  LIN {X 3000.007,Y -1026.300,Z -161.723,A 89.15631,B 0.00000,C 180.00000} ; release
  LIN {X 3000.007,Y -1026.300,Z 138.277,A 89.15631,B 0.00000,C 180.00000} ; retreat
  ; Step 1351, bar 2814
  LIN {X 3750.007,Y -1026.300,Z 1034.024,A 89.15631,B 0.00000,C 180.00000} ; outside
  LIN {X 3750.007,Y -1026.300,Z 88.277,A 89.15631,B 0.00000,C 180.00000} ; preinsert
  LIN {X 3750.007,Y -1026.300,Z -161.723,A 89.15631,B 0.00000,C 180.00000} ; insert
  LIN {X 3750.007,Y -1026.300,Z -161.723,A 89.15631,B 0.00000,C 180.00000} ; release
  LIN {X 3750.007,Y -1026.300,Z 138.277,A 89.15631,B 0.00000,C 180.00000} ; retreat
  ; Step 1352, bar 2817
  LIN {X 4500.007,Y -1026.300,Z 1034.024,A 89.15631,B 0.00000,C 180.00000} ; outside
  LIN {X 4500.007,Y -1026.300,Z 88.277,A 89.15631,B 0.00000,C 180.00000} ; preinsert
  LIN {X 4500.007,Y -1026.300,Z -161.723,A 89.15631,B 0.00000,C 180.00000} ; insert
  LIN {X 4500.007,Y -1026.300,Z -161.723,A 89.15631,B 0.00000,C 180.00000} ; release
  LIN {X 4500.007,Y -1026.300,Z 138.277,A 89.15631,B 0.00000,C 180.00000} ; retreat
  ; Step 1353, bar 2820
  LIN {X 5250.007,Y -1026.300,Z 1034.024,A 89.15631,B 0.00000,C 180.00000} ; outside
  LIN {X 5250.007,Y -1026.300,Z 88.277,A 89.15631,B 0.00000,C 180.00000} ; preinsert
  LIN {X 5250.007,Y -1026.300,Z -161.723,A 89.15631,B 0.00000,C 180.00000} ; insert
  LIN {X 5250.007,Y -1026.300,Z -161.723,A 89.15631,B 0.00000,C 180.00000} ; release
  LIN {X 5250.007,Y -1026.300,Z 138.277,A 89.15631,B 0.00000,C 180.00000} ; retreat
  ; Step 1354, bar 2823
  LIN {X 6000.007,Y -1026.300,Z 1034.024,A 89.15631,B 0.00000,C 180.00000} ; outside
  LIN {X 6000.007,Y -1026.300,Z 88.277,A 89.15631,B 0.00000,C 180.00000} ; preinsert
  LIN {X 6000.007,Y -1026.300,Z -161.723,A 89.15631,B 0.00000,C 180.00000} ; insert
  LIN {X 6000.007,Y -1026.300,Z -161.723,A 89.15631,B 0.00000,C 180.00000} ; release
  LIN {X 6000.007,Y -1026.300,Z 138.277,A 89.15631,B 0.00000,C 180.00000} ; retreat
  ; Step 1355, bar 2826
  LIN {X 6750.007,Y -1026.300,Z 1034.024,A 89.15631,B 0.00000,C 180.00000} ; outside
  LIN {X 6750.007,Y -1026.300,Z 88.277,A 89.15631,B 0.00000,C 180.00000} ; preinsert
  LIN {X 6750.007,Y -1026.300,Z -161.723,A 89.15631,B 0.00000,C 180.00000} ; insert
  LIN {X 6750.007,Y -1026.300,Z -161.723,A 89.15631,B 0.00000,C 180.00000} ; release
  LIN {X 6750.007,Y -1026.300,Z 138.277,A 89.15631,B 0.00000,C 180.00000} ; retreat
  ; Step 1356, bar 2829
  LIN {X 7500.007,Y -1026.300,Z 1034.024,A 89.15631,B 0.00000,C 180.00000} ; outside
  LIN {X 7500.007,Y -1026.300,Z 88.277,A 89.15631,B 0.00000,C 180.00000} ; preinsert
  LIN {X 7500.007,Y -1026.300,Z -161.723,A 89.15631,B 0.00000,C 180.00000} ; insert
  LIN {X 7500.007,Y -1026.300,Z -161.723,A 89.15631,B 0.00000,C 180.00000} ; release
  LIN {X 7500.007,Y -1026.300,Z 138.277,A 89.15631,B 0.00000,C 180.00000} ; retreat
  ; Step 1357, bar 2832
  LIN {X 8250.007,Y -1026.300,Z 1034.024,A 89.15631,B 0.00000,C 180.00000} ; outside
  LIN {X 8250.007,Y -1026.300,Z 88.277,A 89.15631,B 0.00000,C 180.00000} ; preinsert
  LIN {X 8250.007,Y -1026.300,Z -161.723,A 89.15631,B 0.00000,C 180.00000} ; insert
  LIN {X 8250.007,Y -1026.300,Z -161.723,A 89.15631,B 0.00000,C 180.00000} ; release
  LIN {X 8250.007,Y -1026.300,Z 138.277,A 89.15631,B 0.00000,C 180.00000} ; retreat
  ; Step 1358, bar 2835
  LIN {X 9000.007,Y -1026.300,Z 1034.024,A 89.15631,B 0.00000,C 180.00000} ; outside
  LIN {X 9000.007,Y -1026.300,Z 88.277,A 89.15631,B 0.00000,C 180.00000} ; preinsert
  LIN {X 9000.007,Y -1026.300,Z -161.723,A 89.15631,B 0.00000,C 180.00000} ; insert
  LIN {X 9000.007,Y -1026.300,Z -161.723,A 89.15631,B 0.00000,C 180.00000} ; release
  LIN {X 9000.007,Y -1026.300,Z 138.277,A 89.15631,B 0.00000,C 180.00000} ; retreat
  ; Step 1359, bar 2838
  LIN {X 9750.007,Y -1026.300,Z 1034.024,A 89.15631,B 0.00000,C 180.00000} ; outside
  LIN {X 9750.007,Y -1026.300,Z 88.277,A 89.15631,B 0.00000,C 180.00000} ; preinsert
  LIN {X 9750.007,Y -1026.300,Z -161.723,A 89.15631,B 0.00000,C 180.00000} ; insert
  LIN {X 9750.007,Y -1026.300,Z -161.723,A 89.15631,B 0.00000,C 180.00000} ; release
  LIN {X 9750.007,Y -1026.300,Z 138.277,A 89.15631,B 0.00000,C 180.00000} ; retreat
  ; Step 1360, bar 2841
  LIN {X 10500.007,Y -1026.300,Z 1034.024,A 89.15631,B 0.00000,C 180.00000} ; outside
  LIN {X 10500.007,Y -1026.300,Z 88.277,A 89.15631,B 0.00000,C 180.00000} ; preinsert
  LIN {X 10500.007,Y -1026.300,Z -161.723,A 89.15631,B 0.00000,C 180.00000} ; insert
  LIN {X 10500.007,Y -1026.300,Z -161.723,A 89.15631,B 0.00000,C 180.00000} ; release
  LIN {X 10500.007,Y -1026.300,Z 138.277,A 89.15631,B 0.00000,C 180.00000} ; retreat
  ; Step 1361, bar 2844
  LIN {X 11250.007,Y -1026.300,Z 1034.024,A 89.15631,B 0.00000,C 180.00000} ; outside
  LIN {X 11250.007,Y -1026.300,Z 88.277,A 89.15631,B 0.00000,C 180.00000} ; preinsert
  LIN {X 11250.007,Y -1026.300,Z -161.723,A 89.15631,B 0.00000,C 180.00000} ; insert
  LIN {X 11250.007,Y -1026.300,Z -161.723,A 89.15631,B 0.00000,C 180.00000} ; release
  LIN {X 11250.007,Y -1026.300,Z 138.277,A 89.15631,B 0.00000,C 180.00000} ; retreat
  ; Step 1362, bar 2846
  LIN {X 12000.007,Y -1026.300,Z 1034.024,A 89.15631,B 0.00000,C 180.00000} ; outside
  LIN {X 12000.007,Y -1026.300,Z 88.277,A 89.15631,B 0.00000,C 180.00000} ; preinsert
  LIN {X 12000.007,Y -1026.300,Z -161.723,A 89.15631,B 0.00000,C 180.00000} ; insert
  LIN {X 12000.007,Y -1026.300,Z -161.723,A 89.15631,B 0.00000,C 180.00000} ; release
  LIN {X 12000.007,Y -1026.300,Z 138.277,A 89.15631,B 0.00000,C 180.00000} ; retreat
  ; Step 1363, bar 2760
  LIN {X -2250.007,Y -1026.300,Z 1034.024,A 90.84369,B 0.00000,C 180.00000} ; outside
  LIN {X -2250.007,Y -1026.300,Z 88.277,A 90.84369,B 0.00000,C 180.00000} ; preinsert
  LIN {X -2250.007,Y -1026.300,Z -161.723,A 90.84369,B 0.00000,C 180.00000} ; insert
  LIN {X -2250.007,Y -1026.300,Z -161.723,A 90.84369,B 0.00000,C 180.00000} ; release
  LIN {X -2250.007,Y -1026.300,Z 138.277,A 90.84369,B 0.00000,C 180.00000} ; retreat
  ; Step 1364, bar 2763
  LIN {X -3000.007,Y -1026.300,Z 1034.024,A 90.84369,B 0.00000,C 180.00000} ; outside
  LIN {X -3000.007,Y -1026.300,Z 88.277,A 90.84369,B 0.00000,C 180.00000} ; preinsert
  LIN {X -3000.007,Y -1026.300,Z -161.723,A 90.84369,B 0.00000,C 180.00000} ; insert
  LIN {X -3000.007,Y -1026.300,Z -161.723,A 90.84369,B 0.00000,C 180.00000} ; release
  LIN {X -3000.007,Y -1026.300,Z 138.277,A 90.84369,B 0.00000,C 180.00000} ; retreat
  ; Step 1365, bar 2766
  LIN {X -3750.007,Y -1026.300,Z 1034.024,A 90.84369,B 0.00000,C 180.00000} ; outside
  LIN {X -3750.007,Y -1026.300,Z 88.277,A 90.84369,B 0.00000,C 180.00000} ; preinsert
  LIN {X -3750.007,Y -1026.300,Z -161.723,A 90.84369,B 0.00000,C 180.00000} ; insert
  LIN {X -3750.007,Y -1026.300,Z -161.723,A 90.84369,B 0.00000,C 180.00000} ; release
  LIN {X -3750.007,Y -1026.300,Z 138.277,A 90.84369,B 0.00000,C 180.00000} ; retreat
  ; Step 1366, bar 2769
  LIN {X -4500.007,Y -1026.300,Z 1034.024,A 90.84369,B 0.00000,C 180.00000} ; outside
  LIN {X -4500.007,Y -1026.300,Z 88.277,A 90.84369,B 0.00000,C 180.00000} ; preinsert
  LIN {X -4500.007,Y -1026.300,Z -161.723,A 90.84369,B 0.00000,C 180.00000} ; insert
  LIN {X -4500.007,Y -1026.300,Z -161.723,A 90.84369,B 0.00000,C 180.00000} ; release
  LIN {X -4500.007,Y -1026.300,Z 138.277,A 90.84369,B 0.00000,C 180.00000} ; retreat
  ; Step 1367, bar 2772
  LIN {X -5250.007,Y -1026.300,Z 1034.024,A 90.84369,B 0.00000,C 180.00000} ; outside
  LIN {X -5250.007,Y -1026.300,Z 88.277,A 90.84369,B 0.00000,C 180.00000} ; preinsert
  LIN {X -5250.007,Y -1026.300,Z -161.723,A 90.84369,B 0.00000,C 180.00000} ; insert
  LIN {X -5250.007,Y -1026.300,Z -161.723,A 90.84369,B 0.00000,C 180.00000} ; release
  LIN {X -5250.007,Y -1026.300,Z 138.277,A 90.84369,B 0.00000,C 180.00000} ; retreat
  ; Step 1368, bar 2775
  LIN {X -6000.007,Y -1026.300,Z 1034.024,A 90.84369,B 0.00000,C 180.00000} ; outside
  LIN {X -6000.007,Y -1026.300,Z 88.277,A 90.84369,B 0.00000,C 180.00000} ; preinsert
  LIN {X -6000.007,Y -1026.300,Z -161.723,A 90.84369,B 0.00000,C 180.00000} ; insert
  LIN {X -6000.007,Y -1026.300,Z -161.723,A 90.84369,B 0.00000,C 180.00000} ; release
  LIN {X -6000.007,Y -1026.300,Z 138.277,A 90.84369,B 0.00000,C 180.00000} ; retreat
  ; Step 1369, bar 2778
  LIN {X -6750.007,Y -1026.300,Z 1034.024,A 90.84369,B 0.00000,C 180.00000} ; outside
  LIN {X -6750.007,Y -1026.300,Z 88.277,A 90.84369,B 0.00000,C 180.00000} ; preinsert
  LIN {X -6750.007,Y -1026.300,Z -161.723,A 90.84369,B 0.00000,C 180.00000} ; insert
  LIN {X -6750.007,Y -1026.300,Z -161.723,A 90.84369,B 0.00000,C 180.00000} ; release
  LIN {X -6750.007,Y -1026.300,Z 138.277,A 90.84369,B 0.00000,C 180.00000} ; retreat
  ; Step 1370, bar 2781
  LIN {X -7500.007,Y -1026.300,Z 1034.024,A 90.84369,B 0.00000,C 180.00000} ; outside
  LIN {X -7500.007,Y -1026.300,Z 88.277,A 90.84369,B 0.00000,C 180.00000} ; preinsert
  LIN {X -7500.007,Y -1026.300,Z -161.723,A 90.84369,B 0.00000,C 180.00000} ; insert
  LIN {X -7500.007,Y -1026.300,Z -161.723,A 90.84369,B 0.00000,C 180.00000} ; release
  LIN {X -7500.007,Y -1026.300,Z 138.277,A 90.84369,B 0.00000,C 180.00000} ; retreat
  ; Step 1371, bar 2784
  LIN {X -8250.007,Y -1026.300,Z 1034.024,A 90.84369,B 0.00000,C 180.00000} ; outside
  LIN {X -8250.007,Y -1026.300,Z 88.277,A 90.84369,B 0.00000,C 180.00000} ; preinsert
  LIN {X -8250.007,Y -1026.300,Z -161.723,A 90.84369,B 0.00000,C 180.00000} ; insert
  LIN {X -8250.007,Y -1026.300,Z -161.723,A 90.84369,B 0.00000,C 180.00000} ; release
  LIN {X -8250.007,Y -1026.300,Z 138.277,A 90.84369,B 0.00000,C 180.00000} ; retreat
  ; Step 1372, bar 2787
  LIN {X -9000.007,Y -1026.300,Z 1034.024,A 90.84369,B 0.00000,C 180.00000} ; outside
  LIN {X -9000.007,Y -1026.300,Z 88.277,A 90.84369,B 0.00000,C 180.00000} ; preinsert
  LIN {X -9000.007,Y -1026.300,Z -161.723,A 90.84369,B 0.00000,C 180.00000} ; insert
  LIN {X -9000.007,Y -1026.300,Z -161.723,A 90.84369,B 0.00000,C 180.00000} ; release
  LIN {X -9000.007,Y -1026.300,Z 138.277,A 90.84369,B 0.00000,C 180.00000} ; retreat
  ; Step 1373, bar 2790
  LIN {X -9750.007,Y -1026.300,Z 1034.024,A 90.84369,B 0.00000,C 180.00000} ; outside
  LIN {X -9750.007,Y -1026.300,Z 88.277,A 90.84369,B 0.00000,C 180.00000} ; preinsert
  LIN {X -9750.007,Y -1026.300,Z -161.723,A 90.84369,B 0.00000,C 180.00000} ; insert
  LIN {X -9750.007,Y -1026.300,Z -161.723,A 90.84369,B 0.00000,C 180.00000} ; release
  LIN {X -9750.007,Y -1026.300,Z 138.277,A 90.84369,B 0.00000,C 180.00000} ; retreat
  ; Step 1374, bar 2793
  LIN {X -10500.007,Y -1026.300,Z 1034.024,A 90.84369,B 0.00000,C 180.00000} ; outside
  LIN {X -10500.007,Y -1026.300,Z 88.277,A 90.84369,B 0.00000,C 180.00000} ; preinsert
  LIN {X -10500.007,Y -1026.300,Z -161.723,A 90.84369,B 0.00000,C 180.00000} ; insert
  LIN {X -10500.007,Y -1026.300,Z -161.723,A 90.84369,B 0.00000,C 180.00000} ; release
  LIN {X -10500.007,Y -1026.300,Z 138.277,A 90.84369,B 0.00000,C 180.00000} ; retreat
  ; Step 1375, bar 2796
  LIN {X -11250.007,Y -1026.300,Z 1034.024,A 90.84369,B 0.00000,C 180.00000} ; outside
  LIN {X -11250.007,Y -1026.300,Z 88.277,A 90.84369,B 0.00000,C 180.00000} ; preinsert
  LIN {X -11250.007,Y -1026.300,Z -161.723,A 90.84369,B 0.00000,C 180.00000} ; insert
  LIN {X -11250.007,Y -1026.300,Z -161.723,A 90.84369,B 0.00000,C 180.00000} ; release
  LIN {X -11250.007,Y -1026.300,Z 138.277,A 90.84369,B 0.00000,C 180.00000} ; retreat
  ; Step 1376, bar 2798
  LIN {X -12000.007,Y -1026.300,Z 1034.024,A 90.84369,B 0.00000,C 180.00000} ; outside
  LIN {X -12000.007,Y -1026.300,Z 88.277,A 90.84369,B 0.00000,C 180.00000} ; preinsert
  LIN {X -12000.007,Y -1026.300,Z -161.723,A 90.84369,B 0.00000,C 180.00000} ; insert
  LIN {X -12000.007,Y -1026.300,Z -161.723,A 90.84369,B 0.00000,C 180.00000} ; release
  LIN {X -12000.007,Y -1026.300,Z 138.277,A 90.84369,B 0.00000,C 180.00000} ; retreat
  ; Step 1377, bar 2634
  LIN {X -12000.007,Y 1026.300,Z 1034.024,A -90.84369,B 0.00000,C -180.00000} ; outside
  LIN {X -12000.007,Y 1026.300,Z 88.277,A -90.84369,B 0.00000,C -180.00000} ; preinsert
  LIN {X -12000.007,Y 1026.300,Z -161.723,A -90.84369,B 0.00000,C -180.00000} ; insert
  LIN {X -12000.007,Y 1026.300,Z -161.723,A -90.84369,B 0.00000,C -180.00000} ; release
  LIN {X -12000.007,Y 1026.300,Z 138.277,A -90.84369,B 0.00000,C -180.00000} ; retreat
  ; Step 1378, bar 2628
  LIN {X -11250.007,Y 1026.300,Z 1034.024,A -90.84369,B 0.00000,C -180.00000} ; outside
  LIN {X -11250.007,Y 1026.300,Z 88.277,A -90.84369,B 0.00000,C -180.00000} ; preinsert
  LIN {X -11250.007,Y 1026.300,Z -161.723,A -90.84369,B 0.00000,C -180.00000} ; insert
  LIN {X -11250.007,Y 1026.300,Z -161.723,A -90.84369,B 0.00000,C -180.00000} ; release
  LIN {X -11250.007,Y 1026.300,Z 138.277,A -90.84369,B 0.00000,C -180.00000} ; retreat
  ; Step 1379, bar 2621
  LIN {X -10500.007,Y 1026.300,Z 1034.024,A -90.84369,B 0.00000,C -180.00000} ; outside
  LIN {X -10500.007,Y 1026.300,Z 88.277,A -90.84369,B 0.00000,C -180.00000} ; preinsert
  LIN {X -10500.007,Y 1026.300,Z -161.723,A -90.84369,B 0.00000,C -180.00000} ; insert
  LIN {X -10500.007,Y 1026.300,Z -161.723,A -90.84369,B 0.00000,C -180.00000} ; release
  LIN {X -10500.007,Y 1026.300,Z 138.277,A -90.84369,B 0.00000,C -180.00000} ; retreat
  ; Step 1380, bar 2614
  LIN {X -9750.007,Y 1026.300,Z 1034.024,A -90.84369,B 0.00000,C -180.00000} ; outside
  LIN {X -9750.007,Y 1026.300,Z 88.277,A -90.84369,B 0.00000,C -180.00000} ; preinsert
  LIN {X -9750.007,Y 1026.300,Z -161.723,A -90.84369,B 0.00000,C -180.00000} ; insert
  LIN {X -9750.007,Y 1026.300,Z -161.723,A -90.84369,B 0.00000,C -180.00000} ; release
  LIN {X -9750.007,Y 1026.300,Z 138.277,A -90.84369,B 0.00000,C -180.00000} ; retreat
  ; Step 1381, bar 2607
  LIN {X -9000.007,Y 1026.300,Z 1034.024,A -90.84369,B 0.00000,C -180.00000} ; outside
  LIN {X -9000.007,Y 1026.300,Z 88.277,A -90.84369,B 0.00000,C -180.00000} ; preinsert
  LIN {X -9000.007,Y 1026.300,Z -161.723,A -90.84369,B 0.00000,C -180.00000} ; insert
  LIN {X -9000.007,Y 1026.300,Z -161.723,A -90.84369,B 0.00000,C -180.00000} ; release
  LIN {X -9000.007,Y 1026.300,Z 138.277,A -90.84369,B 0.00000,C -180.00000} ; retreat
  ; Step 1382, bar 2600
  LIN {X -8250.007,Y 1026.300,Z 1034.024,A -90.84369,B 0.00000,C -180.00000} ; outside
  LIN {X -8250.007,Y 1026.300,Z 88.277,A -90.84369,B 0.00000,C -180.00000} ; preinsert
  LIN {X -8250.007,Y 1026.300,Z -161.723,A -90.84369,B 0.00000,C -180.00000} ; insert
  LIN {X -8250.007,Y 1026.300,Z -161.723,A -90.84369,B 0.00000,C -180.00000} ; release
  LIN {X -8250.007,Y 1026.300,Z 138.277,A -90.84369,B 0.00000,C -180.00000} ; retreat
  ; Step 1383, bar 2593
  LIN {X -7500.007,Y 1026.300,Z 1034.024,A -90.84369,B 0.00000,C -180.00000} ; outside
  LIN {X -7500.007,Y 1026.300,Z 88.277,A -90.84369,B 0.00000,C -180.00000} ; preinsert
  LIN {X -7500.007,Y 1026.300,Z -161.723,A -90.84369,B 0.00000,C -180.00000} ; insert
  LIN {X -7500.007,Y 1026.300,Z -161.723,A -90.84369,B 0.00000,C -180.00000} ; release
  LIN {X -7500.007,Y 1026.300,Z 138.277,A -90.84369,B 0.00000,C -180.00000} ; retreat
  ; Step 1384, bar 2586
  LIN {X -6750.007,Y 1026.300,Z 1034.024,A -90.84369,B 0.00000,C -180.00000} ; outside
  LIN {X -6750.007,Y 1026.300,Z 88.277,A -90.84369,B 0.00000,C -180.00000} ; preinsert
  LIN {X -6750.007,Y 1026.300,Z -161.723,A -90.84369,B 0.00000,C -180.00000} ; insert
  LIN {X -6750.007,Y 1026.300,Z -161.723,A -90.84369,B 0.00000,C -180.00000} ; release
  LIN {X -6750.007,Y 1026.300,Z 138.277,A -90.84369,B 0.00000,C -180.00000} ; retreat
  ; Step 1385, bar 2579
  LIN {X -6000.007,Y 1026.300,Z 1034.024,A -90.84369,B 0.00000,C -180.00000} ; outside
  LIN {X -6000.007,Y 1026.300,Z 88.277,A -90.84369,B 0.00000,C -180.00000} ; preinsert
  LIN {X -6000.007,Y 1026.300,Z -161.723,A -90.84369,B 0.00000,C -180.00000} ; insert
  LIN {X -6000.007,Y 1026.300,Z -161.723,A -90.84369,B 0.00000,C -180.00000} ; release
  LIN {X -6000.007,Y 1026.300,Z 138.277,A -90.84369,B 0.00000,C -180.00000} ; retreat
  ; Step 1386, bar 2572
  LIN {X -5250.007,Y 1026.300,Z 1034.024,A -90.84369,B 0.00000,C -180.00000} ; outside
  LIN {X -5250.007,Y 1026.300,Z 88.277,A -90.84369,B 0.00000,C -180.00000} ; preinsert
  LIN {X -5250.007,Y 1026.300,Z -161.723,A -90.84369,B 0.00000,C -180.00000} ; insert
  LIN {X -5250.007,Y 1026.300,Z -161.723,A -90.84369,B 0.00000,C -180.00000} ; release
  LIN {X -5250.007,Y 1026.300,Z 138.277,A -90.84369,B 0.00000,C -180.00000} ; retreat
  ; Step 1387, bar 2565
  LIN {X -4500.007,Y 1026.300,Z 1034.024,A -90.84369,B 0.00000,C -180.00000} ; outside
  LIN {X -4500.007,Y 1026.300,Z 88.277,A -90.84369,B 0.00000,C -180.00000} ; preinsert
  LIN {X -4500.007,Y 1026.300,Z -161.723,A -90.84369,B 0.00000,C -180.00000} ; insert
  LIN {X -4500.007,Y 1026.300,Z -161.723,A -90.84369,B 0.00000,C -180.00000} ; release
  LIN {X -4500.007,Y 1026.300,Z 138.277,A -90.84369,B 0.00000,C -180.00000} ; retreat
  ; Step 1388, bar 2558
  LIN {X -3750.007,Y 1026.300,Z 1034.024,A -90.84369,B 0.00000,C -180.00000} ; outside
  LIN {X -3750.007,Y 1026.300,Z 88.277,A -90.84369,B 0.00000,C -180.00000} ; preinsert
  LIN {X -3750.007,Y 1026.300,Z -161.723,A -90.84369,B 0.00000,C -180.00000} ; insert
  LIN {X -3750.007,Y 1026.300,Z -161.723,A -90.84369,B 0.00000,C -180.00000} ; release
  LIN {X -3750.007,Y 1026.300,Z 138.277,A -90.84369,B 0.00000,C -180.00000} ; retreat
  ; Step 1389, bar 2551
  LIN {X -3000.007,Y 1026.300,Z 1034.024,A -90.84369,B 0.00000,C -180.00000} ; outside
  LIN {X -3000.007,Y 1026.300,Z 88.277,A -90.84369,B 0.00000,C -180.00000} ; preinsert
  LIN {X -3000.007,Y 1026.300,Z -161.723,A -90.84369,B 0.00000,C -180.00000} ; insert
  LIN {X -3000.007,Y 1026.300,Z -161.723,A -90.84369,B 0.00000,C -180.00000} ; release
  LIN {X -3000.007,Y 1026.300,Z 138.277,A -90.84369,B 0.00000,C -180.00000} ; retreat
  ; Step 1390, bar 2544
  LIN {X -2250.007,Y 1026.300,Z 1034.024,A -90.84369,B 0.00000,C -180.00000} ; outside
  LIN {X -2250.007,Y 1026.300,Z 88.277,A -90.84369,B 0.00000,C -180.00000} ; preinsert
  LIN {X -2250.007,Y 1026.300,Z -161.723,A -90.84369,B 0.00000,C -180.00000} ; insert
  LIN {X -2250.007,Y 1026.300,Z -161.723,A -90.84369,B 0.00000,C -180.00000} ; release
  LIN {X -2250.007,Y 1026.300,Z 138.277,A -90.84369,B 0.00000,C -180.00000} ; retreat
  ; Step 1391, bar 2537
  LIN {X -1500.007,Y 1026.300,Z 1034.024,A -90.84369,B 0.00000,C -180.00000} ; outside
  LIN {X -1500.007,Y 1026.300,Z 88.277,A -90.84369,B 0.00000,C -180.00000} ; preinsert
  LIN {X -1500.007,Y 1026.300,Z -161.723,A -90.84369,B 0.00000,C -180.00000} ; insert
  LIN {X -1500.007,Y 1026.300,Z -161.723,A -90.84369,B 0.00000,C -180.00000} ; release
  LIN {X -1500.007,Y 1026.300,Z 138.277,A -90.84369,B 0.00000,C -180.00000} ; retreat
  ; Step 1392, bar 2530
  LIN {X -750.007,Y 1026.300,Z 1034.024,A -90.84369,B 0.00000,C -180.00000} ; outside
  LIN {X -750.007,Y 1026.300,Z 88.277,A -90.84369,B 0.00000,C -180.00000} ; preinsert
  LIN {X -750.007,Y 1026.300,Z -161.723,A -90.84369,B 0.00000,C -180.00000} ; insert
  LIN {X -750.007,Y 1026.300,Z -161.723,A -90.84369,B 0.00000,C -180.00000} ; release
  LIN {X -750.007,Y 1026.300,Z 138.277,A -90.84369,B 0.00000,C -180.00000} ; retreat
  ; Step 1393, bar 1971
  LIN {X -0.007,Y 1026.300,Z 1034.024,A -90.84369,B 0.00000,C -180.00000} ; outside
  LIN {X -0.007,Y 1026.300,Z 88.277,A -90.84369,B 0.00000,C -180.00000} ; preinsert
  LIN {X -0.007,Y 1026.300,Z -161.723,A -90.84369,B 0.00000,C -180.00000} ; insert
  LIN {X -0.007,Y 1026.300,Z -161.723,A -90.84369,B 0.00000,C -180.00000} ; release
  LIN {X -0.007,Y 1026.300,Z 138.277,A -90.84369,B 0.00000,C -180.00000} ; retreat
  ; Step 1394, bar 2640
  LIN {X 750.007,Y 1026.300,Z 1034.024,A -89.15631,B 0.00000,C 180.00000} ; outside
  LIN {X 750.007,Y 1026.300,Z 88.277,A -89.15631,B 0.00000,C 180.00000} ; preinsert
  LIN {X 750.007,Y 1026.300,Z -161.723,A -89.15631,B 0.00000,C 180.00000} ; insert
  LIN {X 750.007,Y 1026.300,Z -161.723,A -89.15631,B 0.00000,C 180.00000} ; release
  LIN {X 750.007,Y 1026.300,Z 138.277,A -89.15631,B 0.00000,C 180.00000} ; retreat
  ; Step 1395, bar 2643
  LIN {X 1500.007,Y 1026.300,Z 1034.024,A -89.15631,B 0.00000,C -180.00000} ; outside
  LIN {X 1500.007,Y 1026.300,Z 88.277,A -89.15631,B 0.00000,C -180.00000} ; preinsert
  LIN {X 1500.007,Y 1026.300,Z -161.723,A -89.15631,B 0.00000,C -180.00000} ; insert
  LIN {X 1500.007,Y 1026.300,Z -161.723,A -89.15631,B 0.00000,C -180.00000} ; release
  LIN {X 1500.007,Y 1026.300,Z 138.277,A -89.15631,B 0.00000,C -180.00000} ; retreat
  ; Step 1396, bar 2646
  LIN {X 2250.007,Y 1026.300,Z 1034.024,A -89.15631,B 0.00000,C 180.00000} ; outside
  LIN {X 2250.007,Y 1026.300,Z 88.277,A -89.15631,B 0.00000,C 180.00000} ; preinsert
  LIN {X 2250.007,Y 1026.300,Z -161.723,A -89.15631,B 0.00000,C 180.00000} ; insert
  LIN {X 2250.007,Y 1026.300,Z -161.723,A -89.15631,B 0.00000,C 180.00000} ; release
  LIN {X 2250.007,Y 1026.300,Z 138.277,A -89.15631,B 0.00000,C 180.00000} ; retreat
  ; Step 1397, bar 2649
  LIN {X 3000.007,Y 1026.300,Z 1034.024,A -89.15631,B 0.00000,C 180.00000} ; outside
  LIN {X 3000.007,Y 1026.300,Z 88.277,A -89.15631,B 0.00000,C 180.00000} ; preinsert
  LIN {X 3000.007,Y 1026.300,Z -161.723,A -89.15631,B 0.00000,C 180.00000} ; insert
  LIN {X 3000.007,Y 1026.300,Z -161.723,A -89.15631,B 0.00000,C 180.00000} ; release
  LIN {X 3000.007,Y 1026.300,Z 138.277,A -89.15631,B 0.00000,C 180.00000} ; retreat
  ; Step 1398, bar 2652
  LIN {X 3750.007,Y 1026.300,Z 1034.024,A -89.15631,B 0.00000,C 180.00000} ; outside
  LIN {X 3750.007,Y 1026.300,Z 88.277,A -89.15631,B 0.00000,C 180.00000} ; preinsert
  LIN {X 3750.007,Y 1026.300,Z -161.723,A -89.15631,B 0.00000,C 180.00000} ; insert
  LIN {X 3750.007,Y 1026.300,Z -161.723,A -89.15631,B 0.00000,C 180.00000} ; release
  LIN {X 3750.007,Y 1026.300,Z 138.277,A -89.15631,B 0.00000,C 180.00000} ; retreat
  ; Step 1399, bar 2655
  LIN {X 4500.007,Y 1026.300,Z 1034.024,A -89.15631,B 0.00000,C 180.00000} ; outside
  LIN {X 4500.007,Y 1026.300,Z 88.277,A -89.15631,B 0.00000,C 180.00000} ; preinsert
  LIN {X 4500.007,Y 1026.300,Z -161.723,A -89.15631,B 0.00000,C 180.00000} ; insert
  LIN {X 4500.007,Y 1026.300,Z -161.723,A -89.15631,B 0.00000,C 180.00000} ; release
  LIN {X 4500.007,Y 1026.300,Z 138.277,A -89.15631,B 0.00000,C 180.00000} ; retreat
  ; Step 1400, bar 2658
  LIN {X 5250.007,Y 1026.300,Z 1034.024,A -89.15631,B 0.00000,C 180.00000} ; outside
  LIN {X 5250.007,Y 1026.300,Z 88.277,A -89.15631,B 0.00000,C 180.00000} ; preinsert
  LIN {X 5250.007,Y 1026.300,Z -161.723,A -89.15631,B 0.00000,C 180.00000} ; insert
  LIN {X 5250.007,Y 1026.300,Z -161.723,A -89.15631,B 0.00000,C 180.00000} ; release
  LIN {X 5250.007,Y 1026.300,Z 138.277,A -89.15631,B 0.00000,C 180.00000} ; retreat
  ; Step 1401, bar 2661
  LIN {X 6000.007,Y 1026.300,Z 1034.024,A -89.15631,B 0.00000,C 180.00000} ; outside
  LIN {X 6000.007,Y 1026.300,Z 88.277,A -89.15631,B 0.00000,C 180.00000} ; preinsert
  LIN {X 6000.007,Y 1026.300,Z -161.723,A -89.15631,B 0.00000,C 180.00000} ; insert
  LIN {X 6000.007,Y 1026.300,Z -161.723,A -89.15631,B 0.00000,C 180.00000} ; release
  LIN {X 6000.007,Y 1026.300,Z 138.277,A -89.15631,B 0.00000,C 180.00000} ; retreat
  ; Step 1402, bar 2664
  LIN {X 6750.007,Y 1026.300,Z 1034.024,A -89.15631,B 0.00000,C 180.00000} ; outside
  LIN {X 6750.007,Y 1026.300,Z 88.277,A -89.15631,B 0.00000,C 180.00000} ; preinsert
  LIN {X 6750.007,Y 1026.300,Z -161.723,A -89.15631,B 0.00000,C 180.00000} ; insert
  LIN {X 6750.007,Y 1026.300,Z -161.723,A -89.15631,B 0.00000,C 180.00000} ; release
  LIN {X 6750.007,Y 1026.300,Z 138.277,A -89.15631,B 0.00000,C 180.00000} ; retreat
  ; Step 1403, bar 2667
  LIN {X 7500.007,Y 1026.300,Z 1034.024,A -89.15631,B 0.00000,C 180.00000} ; outside
  LIN {X 7500.007,Y 1026.300,Z 88.277,A -89.15631,B 0.00000,C 180.00000} ; preinsert
  LIN {X 7500.007,Y 1026.300,Z -161.723,A -89.15631,B 0.00000,C 180.00000} ; insert
  LIN {X 7500.007,Y 1026.300,Z -161.723,A -89.15631,B 0.00000,C 180.00000} ; release
  LIN {X 7500.007,Y 1026.300,Z 138.277,A -89.15631,B 0.00000,C 180.00000} ; retreat
  ; Step 1404, bar 2670
  LIN {X 8250.007,Y 1026.300,Z 1034.024,A -89.15631,B 0.00000,C 180.00000} ; outside
  LIN {X 8250.007,Y 1026.300,Z 88.277,A -89.15631,B 0.00000,C 180.00000} ; preinsert
  LIN {X 8250.007,Y 1026.300,Z -161.723,A -89.15631,B 0.00000,C 180.00000} ; insert
  LIN {X 8250.007,Y 1026.300,Z -161.723,A -89.15631,B 0.00000,C 180.00000} ; release
  LIN {X 8250.007,Y 1026.300,Z 138.277,A -89.15631,B 0.00000,C 180.00000} ; retreat
  ; Step 1405, bar 2673
  LIN {X 9000.007,Y 1026.300,Z 1034.024,A -89.15631,B 0.00000,C 180.00000} ; outside
  LIN {X 9000.007,Y 1026.300,Z 88.277,A -89.15631,B 0.00000,C 180.00000} ; preinsert
  LIN {X 9000.007,Y 1026.300,Z -161.723,A -89.15631,B 0.00000,C 180.00000} ; insert
  LIN {X 9000.007,Y 1026.300,Z -161.723,A -89.15631,B 0.00000,C 180.00000} ; release
  LIN {X 9000.007,Y 1026.300,Z 138.277,A -89.15631,B 0.00000,C 180.00000} ; retreat
  ; Step 1406, bar 2676
  LIN {X 9750.007,Y 1026.300,Z 1034.024,A -89.15631,B 0.00000,C 180.00000} ; outside
  LIN {X 9750.007,Y 1026.300,Z 88.277,A -89.15631,B 0.00000,C 180.00000} ; preinsert
  LIN {X 9750.007,Y 1026.300,Z -161.723,A -89.15631,B 0.00000,C 180.00000} ; insert
  LIN {X 9750.007,Y 1026.300,Z -161.723,A -89.15631,B 0.00000,C 180.00000} ; release
  LIN {X 9750.007,Y 1026.300,Z 138.277,A -89.15631,B 0.00000,C 180.00000} ; retreat
  ; Step 1407, bar 2679
  LIN {X 10500.007,Y 1026.300,Z 1034.024,A -89.15631,B 0.00000,C 180.00000} ; outside
  LIN {X 10500.007,Y 1026.300,Z 88.277,A -89.15631,B 0.00000,C 180.00000} ; preinsert
  LIN {X 10500.007,Y 1026.300,Z -161.723,A -89.15631,B 0.00000,C 180.00000} ; insert
  LIN {X 10500.007,Y 1026.300,Z -161.723,A -89.15631,B 0.00000,C 180.00000} ; release
  LIN {X 10500.007,Y 1026.300,Z 138.277,A -89.15631,B 0.00000,C 180.00000} ; retreat
  ; Step 1408, bar 2682
  LIN {X 11250.007,Y 1026.300,Z 1034.024,A -89.15631,B 0.00000,C 180.00000} ; outside
  LIN {X 11250.007,Y 1026.300,Z 88.277,A -89.15631,B 0.00000,C 180.00000} ; preinsert
  LIN {X 11250.007,Y 1026.300,Z -161.723,A -89.15631,B 0.00000,C 180.00000} ; insert
  LIN {X 11250.007,Y 1026.300,Z -161.723,A -89.15631,B 0.00000,C 180.00000} ; release
  LIN {X 11250.007,Y 1026.300,Z 138.277,A -89.15631,B 0.00000,C 180.00000} ; retreat
  ; Step 1409, bar 2684
  LIN {X 12000.007,Y 1026.300,Z 1034.024,A -89.15631,B 0.00000,C 180.00000} ; outside
  LIN {X 12000.007,Y 1026.300,Z 88.277,A -89.15631,B 0.00000,C 180.00000} ; preinsert
  LIN {X 12000.007,Y 1026.300,Z -161.723,A -89.15631,B 0.00000,C 180.00000} ; insert
  LIN {X 12000.007,Y 1026.300,Z -161.723,A -89.15631,B 0.00000,C 180.00000} ; release
  LIN {X 12000.007,Y 1026.300,Z 138.277,A -89.15631,B 0.00000,C 180.00000} ; retreat
  ; Step 1410, bar 277
  LIN {X 0.000,Y 0.000,Z 1139.371,A 0.00000,B 0.00000,C 180.00000} ; outside
  LIN {X 0.000,Y 0.000,Z 193.996,A 0.00000,B 0.00000,C 180.00000} ; preinsert
  LIN {X 0.000,Y 0.000,Z -56.004,A 0.00000,B 0.00000,C 180.00000} ; insert
  LIN {X 0.000,Y 0.000,Z -56.004,A 0.00000,B 0.00000,C 180.00000} ; release
  LIN {X 0.000,Y 0.000,Z 243.996,A 0.00000,B 0.00000,C 180.00000} ; retreat
  ; Step 1411, bar 2526
  LIN {X 16150.007,Y -2866.811,Z 1027.751,A 89.15631,B 0.00000,C 180.00000} ; outside
  LIN {X 16150.007,Y -2866.811,Z 80.465,A 89.15631,B 0.00000,C 180.00000} ; preinsert
  LIN {X 16150.007,Y -2866.811,Z -169.535,A 89.15631,B 0.00000,C 180.00000} ; insert
  LIN {X 16150.007,Y -2866.811,Z -169.535,A 89.15631,B 0.00000,C 180.00000} ; release
  LIN {X 16150.007,Y -2866.811,Z 130.465,A 89.15631,B 0.00000,C 180.00000} ; retreat
  ; Step 1412, bar 2520
  LIN {X 15550.007,Y -2866.811,Z 1027.751,A 89.15631,B 0.00000,C 180.00000} ; outside
  LIN {X 15550.007,Y -2866.811,Z 80.465,A 89.15631,B 0.00000,C 180.00000} ; preinsert
  LIN {X 15550.007,Y -2866.811,Z -169.535,A 89.15631,B 0.00000,C 180.00000} ; insert
  LIN {X 15550.007,Y -2866.811,Z -169.535,A 89.15631,B 0.00000,C 180.00000} ; release
  LIN {X 15550.007,Y -2866.811,Z 130.465,A 89.15631,B 0.00000,C 180.00000} ; retreat
  ; Step 1413, bar 2508
  LIN {X 14350.007,Y -2866.811,Z 1027.751,A 89.15631,B 0.00000,C 180.00000} ; outside
  LIN {X 14350.007,Y -2866.811,Z 80.465,A 89.15631,B 0.00000,C 180.00000} ; preinsert
  LIN {X 14350.007,Y -2866.811,Z -169.535,A 89.15631,B 0.00000,C 180.00000} ; insert
  LIN {X 14350.007,Y -2866.811,Z -169.535,A 89.15631,B 0.00000,C 180.00000} ; release
  LIN {X 14350.007,Y -2866.811,Z 130.465,A 89.15631,B 0.00000,C 180.00000} ; retreat
  ; Step 1414, bar 2514
  LIN {X 14950.007,Y -2866.811,Z 1027.751,A 89.15631,B 0.00000,C 180.00000} ; outside
  LIN {X 14950.007,Y -2866.811,Z 80.465,A 89.15631,B 0.00000,C 180.00000} ; preinsert
  LIN {X 14950.007,Y -2866.811,Z -169.535,A 89.15631,B 0.00000,C 180.00000} ; insert
  LIN {X 14950.007,Y -2866.811,Z -169.535,A 89.15631,B 0.00000,C 180.00000} ; release
  LIN {X 14950.007,Y -2866.811,Z 130.465,A 89.15631,B 0.00000,C 180.00000} ; retreat
  ; Step 1415, bar 2502
  LIN {X 13750.007,Y -2866.811,Z 1027.751,A 89.15631,B 0.00000,C 180.00000} ; outside
  LIN {X 13750.007,Y -2866.811,Z 80.465,A 89.15631,B 0.00000,C 180.00000} ; preinsert
  LIN {X 13750.007,Y -2866.811,Z -169.535,A 89.15631,B 0.00000,C 180.00000} ; insert
  LIN {X 13750.007,Y -2866.811,Z -169.535,A 89.15631,B 0.00000,C 180.00000} ; release
  LIN {X 13750.007,Y -2866.811,Z 130.465,A 89.15631,B 0.00000,C 180.00000} ; retreat
  ; Step 1416, bar 2496
  LIN {X 13150.007,Y -2866.811,Z 1027.751,A 89.15631,B 0.00000,C 180.00000} ; outside
  LIN {X 13150.007,Y -2866.811,Z 80.465,A 89.15631,B 0.00000,C 180.00000} ; preinsert
  LIN {X 13150.007,Y -2866.811,Z -169.535,A 89.15631,B 0.00000,C 180.00000} ; insert
  LIN {X 13150.007,Y -2866.811,Z -169.535,A 89.15631,B 0.00000,C 180.00000} ; release
  LIN {X 13150.007,Y -2866.811,Z 130.465,A 89.15631,B 0.00000,C 180.00000} ; retreat
  ; Step 1417, bar 2490
  LIN {X 12550.007,Y -2866.811,Z 1027.751,A 89.15631,B 0.00000,C 180.00000} ; outside
  LIN {X 12550.007,Y -2866.811,Z 80.465,A 89.15631,B 0.00000,C 180.00000} ; preinsert
  LIN {X 12550.007,Y -2866.811,Z -169.535,A 89.15631,B 0.00000,C 180.00000} ; insert
  LIN {X 12550.007,Y -2866.811,Z -169.535,A 89.15631,B 0.00000,C 180.00000} ; release
  LIN {X 12550.007,Y -2866.811,Z 130.465,A 89.15631,B 0.00000,C 180.00000} ; retreat
  ; Step 1418, bar 2485
  LIN {X 12000.007,Y -2866.811,Z 1027.751,A 89.15631,B 0.00000,C 180.00000} ; outside
  LIN {X 12000.007,Y -2866.811,Z 80.465,A 89.15631,B 0.00000,C 180.00000} ; preinsert
  LIN {X 12000.007,Y -2866.811,Z -169.535,A 89.15631,B 0.00000,C 180.00000} ; insert
  LIN {X 12000.007,Y -2866.811,Z -169.535,A 89.15631,B 0.00000,C 180.00000} ; release
  LIN {X 12000.007,Y -2866.811,Z 130.465,A 89.15631,B 0.00000,C 180.00000} ; retreat
  ; Step 1419, bar 2479
  LIN {X 11250.007,Y -2866.811,Z 1027.751,A 89.15631,B 0.00000,C 180.00000} ; outside
  LIN {X 11250.007,Y -2866.811,Z 80.465,A 89.15631,B 0.00000,C 180.00000} ; preinsert
  LIN {X 11250.007,Y -2866.811,Z -169.535,A 89.15631,B 0.00000,C 180.00000} ; insert
  LIN {X 11250.007,Y -2866.811,Z -169.535,A 89.15631,B 0.00000,C 180.00000} ; release
  LIN {X 11250.007,Y -2866.811,Z 130.465,A 89.15631,B 0.00000,C 180.00000} ; retreat
  ; Step 1420, bar 2473
  LIN {X 10500.007,Y -2866.811,Z 1027.751,A 89.15631,B 0.00000,C 180.00000} ; outside
  LIN {X 10500.007,Y -2866.811,Z 80.465,A 89.15631,B 0.00000,C 180.00000} ; preinsert
  LIN {X 10500.007,Y -2866.811,Z -169.535,A 89.15631,B 0.00000,C 180.00000} ; insert
  LIN {X 10500.007,Y -2866.811,Z -169.535,A 89.15631,B 0.00000,C 180.00000} ; release
  LIN {X 10500.007,Y -2866.811,Z 130.465,A 89.15631,B 0.00000,C 180.00000} ; retreat
  ; Step 1421, bar 2467
  LIN {X 9750.007,Y -2866.811,Z 1027.751,A 89.15631,B 0.00000,C 180.00000} ; outside
  LIN {X 9750.007,Y -2866.811,Z 80.465,A 89.15631,B 0.00000,C 180.00000} ; preinsert
  LIN {X 9750.007,Y -2866.811,Z -169.535,A 89.15631,B 0.00000,C 180.00000} ; insert
  LIN {X 9750.007,Y -2866.811,Z -169.535,A 89.15631,B 0.00000,C 180.00000} ; release
  LIN {X 9750.007,Y -2866.811,Z 130.465,A 89.15631,B 0.00000,C 180.00000} ; retreat
  ; Step 1422, bar 2461
  LIN {X 9000.007,Y -2866.811,Z 1027.751,A 89.15631,B 0.00000,C 180.00000} ; outside
  LIN {X 9000.007,Y -2866.811,Z 80.465,A 89.15631,B 0.00000,C 180.00000} ; preinsert
  LIN {X 9000.007,Y -2866.811,Z -169.535,A 89.15631,B 0.00000,C 180.00000} ; insert
  LIN {X 9000.007,Y -2866.811,Z -169.535,A 89.15631,B 0.00000,C 180.00000} ; release
  LIN {X 9000.007,Y -2866.811,Z 130.465,A 89.15631,B 0.00000,C 180.00000} ; retreat
  ; Step 1423, bar 2455
  LIN {X 8250.007,Y -2866.811,Z 1027.751,A 89.15631,B 0.00000,C 180.00000} ; outside
  LIN {X 8250.007,Y -2866.811,Z 80.465,A 89.15631,B 0.00000,C 180.00000} ; preinsert
  LIN {X 8250.007,Y -2866.811,Z -169.535,A 89.15631,B 0.00000,C 180.00000} ; insert
  LIN {X 8250.007,Y -2866.811,Z -169.535,A 89.15631,B 0.00000,C 180.00000} ; release
  LIN {X 8250.007,Y -2866.811,Z 130.465,A 89.15631,B 0.00000,C 180.00000} ; retreat
  ; Step 1424, bar 2449
  LIN {X 7500.007,Y -2866.811,Z 1027.751,A 89.15631,B 0.00000,C 180.00000} ; outside
  LIN {X 7500.007,Y -2866.811,Z 80.465,A 89.15631,B 0.00000,C 180.00000} ; preinsert
  LIN {X 7500.007,Y -2866.811,Z -169.535,A 89.15631,B 0.00000,C 180.00000} ; insert
  LIN {X 7500.007,Y -2866.811,Z -169.535,A 89.15631,B 0.00000,C 180.00000} ; release
  LIN {X 7500.007,Y -2866.811,Z 130.465,A 89.15631,B 0.00000,C 180.00000} ; retreat
  ; Step 1425, bar 2443
  LIN {X 6750.007,Y -2866.811,Z 1027.751,A 89.15631,B 0.00000,C 180.00000} ; outside
  LIN {X 6750.007,Y -2866.811,Z 80.465,A 89.15631,B 0.00000,C 180.00000} ; preinsert
  LIN {X 6750.007,Y -2866.811,Z -169.535,A 89.15631,B 0.00000,C 180.00000} ; insert
  LIN {X 6750.007,Y -2866.811,Z -169.535,A 89.15631,B 0.00000,C 180.00000} ; release
  LIN {X 6750.007,Y -2866.811,Z 130.465,A 89.15631,B 0.00000,C 180.00000} ; retreat
  ; Step 1426, bar 2437
  LIN {X 6000.007,Y -2866.811,Z 1027.751,A 89.15631,B 0.00000,C 180.00000} ; outside
  LIN {X 6000.007,Y -2866.811,Z 80.465,A 89.15631,B 0.00000,C 180.00000} ; preinsert
  LIN {X 6000.007,Y -2866.811,Z -169.535,A 89.15631,B 0.00000,C 180.00000} ; insert
  LIN {X 6000.007,Y -2866.811,Z -169.535,A 89.15631,B 0.00000,C 180.00000} ; release
  LIN {X 6000.007,Y -2866.811,Z 130.465,A 89.15631,B 0.00000,C 180.00000} ; retreat
  ; Step 1427, bar 2431
  LIN {X 5250.007,Y -2866.811,Z 1027.751,A 89.15631,B 0.00000,C 180.00000} ; outside
  LIN {X 5250.007,Y -2866.811,Z 80.465,A 89.15631,B 0.00000,C 180.00000} ; preinsert
  LIN {X 5250.007,Y -2866.811,Z -169.535,A 89.15631,B 0.00000,C 180.00000} ; insert
  LIN {X 5250.007,Y -2866.811,Z -169.535,A 89.15631,B 0.00000,C 180.00000} ; release
  LIN {X 5250.007,Y -2866.811,Z 130.465,A 89.15631,B 0.00000,C 180.00000} ; retreat
  ; Step 1428, bar 2425
  LIN {X 4500.007,Y -2866.811,Z 1027.751,A 89.15631,B 0.00000,C 180.00000} ; outside
  LIN {X 4500.007,Y -2866.811,Z 80.465,A 89.15631,B 0.00000,C 180.00000} ; preinsert
  LIN {X 4500.007,Y -2866.811,Z -169.535,A 89.15631,B 0.00000,C 180.00000} ; insert
  LIN {X 4500.007,Y -2866.811,Z -169.535,A 89.15631,B 0.00000,C 180.00000} ; release
  LIN {X 4500.007,Y -2866.811,Z 130.465,A 89.15631,B 0.00000,C 180.00000} ; retreat
  ; Step 1429, bar 2419
  LIN {X 3750.007,Y -2866.811,Z 1027.751,A 89.15631,B 0.00000,C 180.00000} ; outside
  LIN {X 3750.007,Y -2866.811,Z 80.465,A 89.15631,B 0.00000,C 180.00000} ; preinsert
  LIN {X 3750.007,Y -2866.811,Z -169.535,A 89.15631,B 0.00000,C 180.00000} ; insert
  LIN {X 3750.007,Y -2866.811,Z -169.535,A 89.15631,B 0.00000,C 180.00000} ; release
  LIN {X 3750.007,Y -2866.811,Z 130.465,A 89.15631,B 0.00000,C 180.00000} ; retreat
  ; Step 1430, bar 2413
  LIN {X 3000.007,Y -2866.811,Z 1027.751,A 89.15631,B 0.00000,C 180.00000} ; outside
  LIN {X 3000.007,Y -2866.811,Z 80.465,A 89.15631,B 0.00000,C 180.00000} ; preinsert
  LIN {X 3000.007,Y -2866.811,Z -169.535,A 89.15631,B 0.00000,C 180.00000} ; insert
  LIN {X 3000.007,Y -2866.811,Z -169.535,A 89.15631,B 0.00000,C 180.00000} ; release
  LIN {X 3000.007,Y -2866.811,Z 130.465,A 89.15631,B 0.00000,C 180.00000} ; retreat
  ; Step 1431, bar 2407
  LIN {X 2250.007,Y -2866.811,Z 1027.751,A 89.15631,B 0.00000,C 180.00000} ; outside
  LIN {X 2250.007,Y -2866.811,Z 80.465,A 89.15631,B 0.00000,C 180.00000} ; preinsert
  LIN {X 2250.007,Y -2866.811,Z -169.535,A 89.15631,B 0.00000,C 180.00000} ; insert
  LIN {X 2250.007,Y -2866.811,Z -169.535,A 89.15631,B 0.00000,C 180.00000} ; release
  LIN {X 2250.007,Y -2866.811,Z 130.465,A 89.15631,B 0.00000,C 180.00000} ; retreat
  ; Step 1432, bar 2401
  LIN {X 1500.007,Y -2866.811,Z 1027.751,A 89.15631,B 0.00000,C 180.00000} ; outside
  LIN {X 1500.007,Y -2866.811,Z 80.465,A 89.15631,B 0.00000,C 180.00000} ; preinsert
  LIN {X 1500.007,Y -2866.811,Z -169.535,A 89.15631,B 0.00000,C 180.00000} ; insert
  LIN {X 1500.007,Y -2866.811,Z -169.535,A 89.15631,B 0.00000,C 180.00000} ; release
  LIN {X 1500.007,Y -2866.811,Z 130.465,A 89.15631,B 0.00000,C 180.00000} ; retreat
  ; Step 1433, bar 2395
  LIN {X 750.007,Y -2866.811,Z 1027.751,A 89.15631,B 0.00000,C 180.00000} ; outside
  LIN {X 750.007,Y -2866.811,Z 80.465,A 89.15631,B 0.00000,C 180.00000} ; preinsert
  LIN {X 750.007,Y -2866.811,Z -169.535,A 89.15631,B 0.00000,C 180.00000} ; insert
  LIN {X 750.007,Y -2866.811,Z -169.535,A 89.15631,B 0.00000,C 180.00000} ; release
  LIN {X 750.007,Y -2866.811,Z 130.465,A 89.15631,B 0.00000,C 180.00000} ; retreat
  ; Step 1434, bar 2251
  LIN {X -0.007,Y -2866.811,Z 1027.751,A 90.84369,B 0.00000,C -180.00000} ; outside
  LIN {X -0.007,Y -2866.811,Z 80.465,A 90.84369,B 0.00000,C -180.00000} ; preinsert
  LIN {X -0.007,Y -2866.811,Z -169.535,A 90.84369,B 0.00000,C -180.00000} ; insert
  LIN {X -0.007,Y -2866.811,Z -169.535,A 90.84369,B 0.00000,C -180.00000} ; release
  LIN {X -0.007,Y -2866.811,Z 130.465,A 90.84369,B 0.00000,C -180.00000} ; retreat
  ; Step 1435, bar 2257
  LIN {X -750.007,Y -2866.811,Z 1027.751,A 90.84369,B 0.00000,C 180.00000} ; outside
  LIN {X -750.007,Y -2866.811,Z 80.465,A 90.84369,B 0.00000,C 180.00000} ; preinsert
  LIN {X -750.007,Y -2866.811,Z -169.535,A 90.84369,B 0.00000,C 180.00000} ; insert
  LIN {X -750.007,Y -2866.811,Z -169.535,A 90.84369,B 0.00000,C 180.00000} ; release
  LIN {X -750.007,Y -2866.811,Z 130.465,A 90.84369,B 0.00000,C 180.00000} ; retreat
  ; Step 1436, bar 2263
  LIN {X -1500.007,Y -2866.811,Z 1027.751,A 90.84369,B 0.00000,C 180.00000} ; outside
  LIN {X -1500.007,Y -2866.811,Z 80.465,A 90.84369,B 0.00000,C 180.00000} ; preinsert
  LIN {X -1500.007,Y -2866.811,Z -169.535,A 90.84369,B 0.00000,C 180.00000} ; insert
  LIN {X -1500.007,Y -2866.811,Z -169.535,A 90.84369,B 0.00000,C 180.00000} ; release
  LIN {X -1500.007,Y -2866.811,Z 130.465,A 90.84369,B 0.00000,C 180.00000} ; retreat
  ; Step 1437, bar 2269
  LIN {X -2250.007,Y -2866.811,Z 1027.751,A 90.84369,B 0.00000,C -180.00000} ; outside
  LIN {X -2250.007,Y -2866.811,Z 80.465,A 90.84369,B 0.00000,C -180.00000} ; preinsert
  LIN {X -2250.007,Y -2866.811,Z -169.535,A 90.84369,B 0.00000,C -180.00000} ; insert
  LIN {X -2250.007,Y -2866.811,Z -169.535,A 90.84369,B 0.00000,C -180.00000} ; release
  LIN {X -2250.007,Y -2866.811,Z 130.465,A 90.84369,B 0.00000,C -180.00000} ; retreat
  ; Step 1438, bar 2275
  LIN {X -3000.007,Y -2866.811,Z 1027.751,A 90.84369,B 0.00000,C -180.00000} ; outside
  LIN {X -3000.007,Y -2866.811,Z 80.465,A 90.84369,B 0.00000,C -180.00000} ; preinsert
  LIN {X -3000.007,Y -2866.811,Z -169.535,A 90.84369,B 0.00000,C -180.00000} ; insert
  LIN {X -3000.007,Y -2866.811,Z -169.535,A 90.84369,B 0.00000,C -180.00000} ; release
  LIN {X -3000.007,Y -2866.811,Z 130.465,A 90.84369,B 0.00000,C -180.00000} ; retreat
  ; Step 1439, bar 2281
  LIN {X -3750.007,Y -2866.811,Z 1027.751,A 90.84369,B 0.00000,C -180.00000} ; outside
  LIN {X -3750.007,Y -2866.811,Z 80.465,A 90.84369,B 0.00000,C -180.00000} ; preinsert
  LIN {X -3750.007,Y -2866.811,Z -169.535,A 90.84369,B 0.00000,C -180.00000} ; insert
  LIN {X -3750.007,Y -2866.811,Z -169.535,A 90.84369,B 0.00000,C -180.00000} ; release
  LIN {X -3750.007,Y -2866.811,Z 130.465,A 90.84369,B 0.00000,C -180.00000} ; retreat
  ; Step 1440, bar 2287
  LIN {X -4500.007,Y -2866.811,Z 1027.751,A 90.84369,B 0.00000,C -180.00000} ; outside
  LIN {X -4500.007,Y -2866.811,Z 80.465,A 90.84369,B 0.00000,C -180.00000} ; preinsert
  LIN {X -4500.007,Y -2866.811,Z -169.535,A 90.84369,B 0.00000,C -180.00000} ; insert
  LIN {X -4500.007,Y -2866.811,Z -169.535,A 90.84369,B 0.00000,C -180.00000} ; release
  LIN {X -4500.007,Y -2866.811,Z 130.465,A 90.84369,B 0.00000,C -180.00000} ; retreat
  ; Step 1441, bar 2293
  LIN {X -5250.007,Y -2866.811,Z 1027.751,A 90.84369,B 0.00000,C -180.00000} ; outside
  LIN {X -5250.007,Y -2866.811,Z 80.465,A 90.84369,B 0.00000,C -180.00000} ; preinsert
  LIN {X -5250.007,Y -2866.811,Z -169.535,A 90.84369,B 0.00000,C -180.00000} ; insert
  LIN {X -5250.007,Y -2866.811,Z -169.535,A 90.84369,B 0.00000,C -180.00000} ; release
  LIN {X -5250.007,Y -2866.811,Z 130.465,A 90.84369,B 0.00000,C -180.00000} ; retreat
  ; Step 1442, bar 2299
  LIN {X -6000.007,Y -2866.811,Z 1027.751,A 90.84369,B 0.00000,C -180.00000} ; outside
  LIN {X -6000.007,Y -2866.811,Z 80.465,A 90.84369,B 0.00000,C -180.00000} ; preinsert
  LIN {X -6000.007,Y -2866.811,Z -169.535,A 90.84369,B 0.00000,C -180.00000} ; insert
  LIN {X -6000.007,Y -2866.811,Z -169.535,A 90.84369,B 0.00000,C -180.00000} ; release
  LIN {X -6000.007,Y -2866.811,Z 130.465,A 90.84369,B 0.00000,C -180.00000} ; retreat
  ; Step 1443, bar 2305
  LIN {X -6750.007,Y -2866.811,Z 1027.751,A 90.84369,B 0.00000,C -180.00000} ; outside
  LIN {X -6750.007,Y -2866.811,Z 80.465,A 90.84369,B 0.00000,C -180.00000} ; preinsert
  LIN {X -6750.007,Y -2866.811,Z -169.535,A 90.84369,B 0.00000,C -180.00000} ; insert
  LIN {X -6750.007,Y -2866.811,Z -169.535,A 90.84369,B 0.00000,C -180.00000} ; release
  LIN {X -6750.007,Y -2866.811,Z 130.465,A 90.84369,B 0.00000,C -180.00000} ; retreat
  ; Step 1444, bar 2311
  LIN {X -7500.007,Y -2866.811,Z 1027.751,A 90.84369,B 0.00000,C -180.00000} ; outside
  LIN {X -7500.007,Y -2866.811,Z 80.465,A 90.84369,B 0.00000,C -180.00000} ; preinsert
  LIN {X -7500.007,Y -2866.811,Z -169.535,A 90.84369,B 0.00000,C -180.00000} ; insert
  LIN {X -7500.007,Y -2866.811,Z -169.535,A 90.84369,B 0.00000,C -180.00000} ; release
  LIN {X -7500.007,Y -2866.811,Z 130.465,A 90.84369,B 0.00000,C -180.00000} ; retreat
  ; Step 1445, bar 2317
  LIN {X -8250.007,Y -2866.811,Z 1027.751,A 90.84369,B 0.00000,C 180.00000} ; outside
  LIN {X -8250.007,Y -2866.811,Z 80.465,A 90.84369,B 0.00000,C 180.00000} ; preinsert
  LIN {X -8250.007,Y -2866.811,Z -169.535,A 90.84369,B 0.00000,C 180.00000} ; insert
  LIN {X -8250.007,Y -2866.811,Z -169.535,A 90.84369,B 0.00000,C 180.00000} ; release
  LIN {X -8250.007,Y -2866.811,Z 130.465,A 90.84369,B 0.00000,C 180.00000} ; retreat
  ; Step 1446, bar 2323
  LIN {X -9000.007,Y -2866.811,Z 1027.751,A 90.84369,B 0.00000,C 180.00000} ; outside
  LIN {X -9000.007,Y -2866.811,Z 80.465,A 90.84369,B 0.00000,C 180.00000} ; preinsert
  LIN {X -9000.007,Y -2866.811,Z -169.535,A 90.84369,B 0.00000,C 180.00000} ; insert
  LIN {X -9000.007,Y -2866.811,Z -169.535,A 90.84369,B 0.00000,C 180.00000} ; release
  LIN {X -9000.007,Y -2866.811,Z 130.465,A 90.84369,B 0.00000,C 180.00000} ; retreat
  ; Step 1447, bar 2329
  LIN {X -9750.007,Y -2866.811,Z 1027.751,A 90.84369,B 0.00000,C 180.00000} ; outside
  LIN {X -9750.007,Y -2866.811,Z 80.465,A 90.84369,B 0.00000,C 180.00000} ; preinsert
  LIN {X -9750.007,Y -2866.811,Z -169.535,A 90.84369,B 0.00000,C 180.00000} ; insert
  LIN {X -9750.007,Y -2866.811,Z -169.535,A 90.84369,B 0.00000,C 180.00000} ; release
  LIN {X -9750.007,Y -2866.811,Z 130.465,A 90.84369,B 0.00000,C 180.00000} ; retreat
  ; Step 1448, bar 2335
  LIN {X -10500.007,Y -2866.811,Z 1027.751,A 90.84369,B 0.00000,C 180.00000} ; outside
  LIN {X -10500.007,Y -2866.811,Z 80.465,A 90.84369,B 0.00000,C 180.00000} ; preinsert
  LIN {X -10500.007,Y -2866.811,Z -169.535,A 90.84369,B 0.00000,C 180.00000} ; insert
  LIN {X -10500.007,Y -2866.811,Z -169.535,A 90.84369,B 0.00000,C 180.00000} ; release
  LIN {X -10500.007,Y -2866.811,Z 130.465,A 90.84369,B 0.00000,C 180.00000} ; retreat
  ; Step 1449, bar 2341
  LIN {X -11250.007,Y -2866.811,Z 1027.751,A 90.84369,B 0.00000,C 180.00000} ; outside
  LIN {X -11250.007,Y -2866.811,Z 80.465,A 90.84369,B 0.00000,C 180.00000} ; preinsert
  LIN {X -11250.007,Y -2866.811,Z -169.535,A 90.84369,B 0.00000,C 180.00000} ; insert
  LIN {X -11250.007,Y -2866.811,Z -169.535,A 90.84369,B 0.00000,C 180.00000} ; release
  LIN {X -11250.007,Y -2866.811,Z 130.465,A 90.84369,B 0.00000,C 180.00000} ; retreat
  ; Step 1450, bar 2347
  LIN {X -12000.007,Y -2866.811,Z 1027.751,A 90.84369,B 0.00000,C 180.00000} ; outside
  LIN {X -12000.007,Y -2866.811,Z 80.465,A 90.84369,B 0.00000,C 180.00000} ; preinsert
  LIN {X -12000.007,Y -2866.811,Z -169.535,A 90.84369,B 0.00000,C 180.00000} ; insert
  LIN {X -12000.007,Y -2866.811,Z -169.535,A 90.84369,B 0.00000,C 180.00000} ; release
  LIN {X -12000.007,Y -2866.811,Z 130.465,A 90.84369,B 0.00000,C 180.00000} ; retreat
  ; Step 1451, bar 2352
  LIN {X -12550.007,Y -2866.811,Z 1027.751,A 90.84369,B 0.00000,C 180.00000} ; outside
  LIN {X -12550.007,Y -2866.811,Z 80.465,A 90.84369,B 0.00000,C 180.00000} ; preinsert
  LIN {X -12550.007,Y -2866.811,Z -169.535,A 90.84369,B 0.00000,C 180.00000} ; insert
  LIN {X -12550.007,Y -2866.811,Z -169.535,A 90.84369,B 0.00000,C 180.00000} ; release
  LIN {X -12550.007,Y -2866.811,Z 130.465,A 90.84369,B 0.00000,C 180.00000} ; retreat
  ; Step 1452, bar 2358
  LIN {X -13150.007,Y -2866.811,Z 1027.751,A 90.84369,B 0.00000,C 180.00000} ; outside
  LIN {X -13150.007,Y -2866.811,Z 80.465,A 90.84369,B 0.00000,C 180.00000} ; preinsert
  LIN {X -13150.007,Y -2866.811,Z -169.535,A 90.84369,B 0.00000,C 180.00000} ; insert
  LIN {X -13150.007,Y -2866.811,Z -169.535,A 90.84369,B 0.00000,C 180.00000} ; release
  LIN {X -13150.007,Y -2866.811,Z 130.465,A 90.84369,B 0.00000,C 180.00000} ; retreat
  ; Step 1453, bar 2364
  LIN {X -13750.007,Y -2866.811,Z 1027.751,A 90.84369,B 0.00000,C 180.00000} ; outside
  LIN {X -13750.007,Y -2866.811,Z 80.465,A 90.84369,B 0.00000,C 180.00000} ; preinsert
  LIN {X -13750.007,Y -2866.811,Z -169.535,A 90.84369,B 0.00000,C 180.00000} ; insert
  LIN {X -13750.007,Y -2866.811,Z -169.535,A 90.84369,B 0.00000,C 180.00000} ; release
  LIN {X -13750.007,Y -2866.811,Z 130.465,A 90.84369,B 0.00000,C 180.00000} ; retreat
  ; Step 1454, bar 2376
  LIN {X -14950.007,Y -2866.811,Z 1027.751,A 90.84369,B 0.00000,C 180.00000} ; outside
  LIN {X -14950.007,Y -2866.811,Z 80.465,A 90.84369,B 0.00000,C 180.00000} ; preinsert
  LIN {X -14950.007,Y -2866.811,Z -169.535,A 90.84369,B 0.00000,C 180.00000} ; insert
  LIN {X -14950.007,Y -2866.811,Z -169.535,A 90.84369,B 0.00000,C 180.00000} ; release
  LIN {X -14950.007,Y -2866.811,Z 130.465,A 90.84369,B 0.00000,C 180.00000} ; retreat
  ; Step 1455, bar 2370
  LIN {X -14350.007,Y -2866.811,Z 1027.751,A 90.84369,B 0.00000,C 180.00000} ; outside
  LIN {X -14350.007,Y -2866.811,Z 80.465,A 90.84369,B 0.00000,C 180.00000} ; preinsert
  LIN {X -14350.007,Y -2866.811,Z -169.535,A 90.84369,B 0.00000,C 180.00000} ; insert
  LIN {X -14350.007,Y -2866.811,Z -169.535,A 90.84369,B 0.00000,C 180.00000} ; release
  LIN {X -14350.007,Y -2866.811,Z 130.465,A 90.84369,B 0.00000,C 180.00000} ; retreat
  ; Step 1456, bar 2382
  LIN {X -15550.007,Y -2866.811,Z 1027.751,A 90.84369,B 0.00000,C 180.00000} ; outside
  LIN {X -15550.007,Y -2866.811,Z 80.465,A 90.84369,B 0.00000,C 180.00000} ; preinsert
  LIN {X -15550.007,Y -2866.811,Z -169.535,A 90.84369,B 0.00000,C 180.00000} ; insert
  LIN {X -15550.007,Y -2866.811,Z -169.535,A 90.84369,B 0.00000,C 180.00000} ; release
  LIN {X -15550.007,Y -2866.811,Z 130.465,A 90.84369,B 0.00000,C 180.00000} ; retreat
  ; Step 1457, bar 2388
  LIN {X -16150.007,Y -2866.811,Z 1027.751,A 90.84369,B 0.00000,C 180.00000} ; outside
  LIN {X -16150.007,Y -2866.811,Z 80.465,A 90.84369,B 0.00000,C 180.00000} ; preinsert
  LIN {X -16150.007,Y -2866.811,Z -169.535,A 90.84369,B 0.00000,C 180.00000} ; insert
  LIN {X -16150.007,Y -2866.811,Z -169.535,A 90.84369,B 0.00000,C 180.00000} ; release
  LIN {X -16150.007,Y -2866.811,Z 130.465,A 90.84369,B 0.00000,C 180.00000} ; retreat
  ; Step 1458, bar 2109
  LIN {X -16150.007,Y 2866.811,Z 1027.751,A -90.84369,B 0.00000,C -180.00000} ; outside
  LIN {X -16150.007,Y 2866.811,Z 80.465,A -90.84369,B 0.00000,C -180.00000} ; preinsert
  LIN {X -16150.007,Y 2866.811,Z -169.535,A -90.84369,B 0.00000,C -180.00000} ; insert
  LIN {X -16150.007,Y 2866.811,Z -169.535,A -90.84369,B 0.00000,C -180.00000} ; release
  LIN {X -16150.007,Y 2866.811,Z 130.465,A -90.84369,B 0.00000,C -180.00000} ; retreat
  ; Step 1459, bar 2103
  LIN {X -15550.007,Y 2866.811,Z 1027.751,A -90.84369,B 0.00000,C -180.00000} ; outside
  LIN {X -15550.007,Y 2866.811,Z 80.465,A -90.84369,B 0.00000,C -180.00000} ; preinsert
  LIN {X -15550.007,Y 2866.811,Z -169.535,A -90.84369,B 0.00000,C -180.00000} ; insert
  LIN {X -15550.007,Y 2866.811,Z -169.535,A -90.84369,B 0.00000,C -180.00000} ; release
  LIN {X -15550.007,Y 2866.811,Z 130.465,A -90.84369,B 0.00000,C -180.00000} ; retreat
  ; Step 1460, bar 2097
  LIN {X -14950.007,Y 2866.811,Z 1027.751,A -90.84369,B 0.00000,C -180.00000} ; outside
  LIN {X -14950.007,Y 2866.811,Z 80.465,A -90.84369,B 0.00000,C -180.00000} ; preinsert
  LIN {X -14950.007,Y 2866.811,Z -169.535,A -90.84369,B 0.00000,C -180.00000} ; insert
  LIN {X -14950.007,Y 2866.811,Z -169.535,A -90.84369,B 0.00000,C -180.00000} ; release
  LIN {X -14950.007,Y 2866.811,Z 130.465,A -90.84369,B 0.00000,C -180.00000} ; retreat
  ; Step 1461, bar 2091
  LIN {X -14350.007,Y 2866.811,Z 1027.751,A -90.84369,B 0.00000,C -180.00000} ; outside
  LIN {X -14350.007,Y 2866.811,Z 80.465,A -90.84369,B 0.00000,C -180.00000} ; preinsert
  LIN {X -14350.007,Y 2866.811,Z -169.535,A -90.84369,B 0.00000,C -180.00000} ; insert
  LIN {X -14350.007,Y 2866.811,Z -169.535,A -90.84369,B 0.00000,C -180.00000} ; release
  LIN {X -14350.007,Y 2866.811,Z 130.465,A -90.84369,B 0.00000,C -180.00000} ; retreat
  ; Step 1462, bar 2085
  LIN {X -13750.007,Y 2866.811,Z 1027.751,A -90.84369,B 0.00000,C -180.00000} ; outside
  LIN {X -13750.007,Y 2866.811,Z 80.465,A -90.84369,B 0.00000,C -180.00000} ; preinsert
  LIN {X -13750.007,Y 2866.811,Z -169.535,A -90.84369,B 0.00000,C -180.00000} ; insert
  LIN {X -13750.007,Y 2866.811,Z -169.535,A -90.84369,B 0.00000,C -180.00000} ; release
  LIN {X -13750.007,Y 2866.811,Z 130.465,A -90.84369,B 0.00000,C -180.00000} ; retreat
  ; Step 1463, bar 2079
  LIN {X -13150.007,Y 2866.811,Z 1027.751,A -90.84369,B 0.00000,C -180.00000} ; outside
  LIN {X -13150.007,Y 2866.811,Z 80.465,A -90.84369,B 0.00000,C -180.00000} ; preinsert
  LIN {X -13150.007,Y 2866.811,Z -169.535,A -90.84369,B 0.00000,C -180.00000} ; insert
  LIN {X -13150.007,Y 2866.811,Z -169.535,A -90.84369,B 0.00000,C -180.00000} ; release
  LIN {X -13150.007,Y 2866.811,Z 130.465,A -90.84369,B 0.00000,C -180.00000} ; retreat
  ; Step 1464, bar 2073
  LIN {X -12550.007,Y 2866.811,Z 1027.751,A -90.84369,B 0.00000,C -180.00000} ; outside
  LIN {X -12550.007,Y 2866.811,Z 80.465,A -90.84369,B 0.00000,C -180.00000} ; preinsert
  LIN {X -12550.007,Y 2866.811,Z -169.535,A -90.84369,B 0.00000,C -180.00000} ; insert
  LIN {X -12550.007,Y 2866.811,Z -169.535,A -90.84369,B 0.00000,C -180.00000} ; release
  LIN {X -12550.007,Y 2866.811,Z 130.465,A -90.84369,B 0.00000,C -180.00000} ; retreat
  ; Step 1465, bar 2068
  LIN {X -12000.007,Y 2866.811,Z 1027.751,A -90.84369,B 0.00000,C -180.00000} ; outside
  LIN {X -12000.007,Y 2866.811,Z 80.465,A -90.84369,B 0.00000,C -180.00000} ; preinsert
  LIN {X -12000.007,Y 2866.811,Z -169.535,A -90.84369,B 0.00000,C -180.00000} ; insert
  LIN {X -12000.007,Y 2866.811,Z -169.535,A -90.84369,B 0.00000,C -180.00000} ; release
  LIN {X -12000.007,Y 2866.811,Z 130.465,A -90.84369,B 0.00000,C -180.00000} ; retreat
  ; Step 1466, bar 2062
  LIN {X -11250.007,Y 2866.811,Z 1027.751,A -90.84369,B 0.00000,C -180.00000} ; outside
  LIN {X -11250.007,Y 2866.811,Z 80.465,A -90.84369,B 0.00000,C -180.00000} ; preinsert
  LIN {X -11250.007,Y 2866.811,Z -169.535,A -90.84369,B 0.00000,C -180.00000} ; insert
  LIN {X -11250.007,Y 2866.811,Z -169.535,A -90.84369,B 0.00000,C -180.00000} ; release
  LIN {X -11250.007,Y 2866.811,Z 130.465,A -90.84369,B 0.00000,C -180.00000} ; retreat
  ; Step 1467, bar 2056
  LIN {X -10500.007,Y 2866.811,Z 1027.751,A -90.84369,B 0.00000,C -180.00000} ; outside
  LIN {X -10500.007,Y 2866.811,Z 80.465,A -90.84369,B 0.00000,C -180.00000} ; preinsert
  LIN {X -10500.007,Y 2866.811,Z -169.535,A -90.84369,B 0.00000,C -180.00000} ; insert
  LIN {X -10500.007,Y 2866.811,Z -169.535,A -90.84369,B 0.00000,C -180.00000} ; release
  LIN {X -10500.007,Y 2866.811,Z 130.465,A -90.84369,B 0.00000,C -180.00000} ; retreat
  ; Step 1468, bar 2050
  LIN {X -9750.007,Y 2866.811,Z 1027.751,A -90.84369,B 0.00000,C -180.00000} ; outside
  LIN {X -9750.007,Y 2866.811,Z 80.465,A -90.84369,B 0.00000,C -180.00000} ; preinsert
  LIN {X -9750.007,Y 2866.811,Z -169.535,A -90.84369,B 0.00000,C -180.00000} ; insert
  LIN {X -9750.007,Y 2866.811,Z -169.535,A -90.84369,B 0.00000,C -180.00000} ; release
  LIN {X -9750.007,Y 2866.811,Z 130.465,A -90.84369,B 0.00000,C -180.00000} ; retreat
  ; Step 1469, bar 2044
  LIN {X -9000.007,Y 2866.811,Z 1027.751,A -90.84369,B 0.00000,C -180.00000} ; outside
  LIN {X -9000.007,Y 2866.811,Z 80.465,A -90.84369,B 0.00000,C -180.00000} ; preinsert
  LIN {X -9000.007,Y 2866.811,Z -169.535,A -90.84369,B 0.00000,C -180.00000} ; insert
  LIN {X -9000.007,Y 2866.811,Z -169.535,A -90.84369,B 0.00000,C -180.00000} ; release
  LIN {X -9000.007,Y 2866.811,Z 130.465,A -90.84369,B 0.00000,C -180.00000} ; retreat
  ; Step 1470, bar 2038
  LIN {X -8250.007,Y 2866.811,Z 1027.751,A -90.84369,B 0.00000,C -180.00000} ; outside
  LIN {X -8250.007,Y 2866.811,Z 80.465,A -90.84369,B 0.00000,C -180.00000} ; preinsert
  LIN {X -8250.007,Y 2866.811,Z -169.535,A -90.84369,B 0.00000,C -180.00000} ; insert
  LIN {X -8250.007,Y 2866.811,Z -169.535,A -90.84369,B 0.00000,C -180.00000} ; release
  LIN {X -8250.007,Y 2866.811,Z 130.465,A -90.84369,B 0.00000,C -180.00000} ; retreat
  ; Step 1471, bar 2032
  LIN {X -7500.007,Y 2866.811,Z 1027.751,A -90.84369,B 0.00000,C 180.00000} ; outside
  LIN {X -7500.007,Y 2866.811,Z 80.465,A -90.84369,B 0.00000,C 180.00000} ; preinsert
  LIN {X -7500.007,Y 2866.811,Z -169.535,A -90.84369,B 0.00000,C 180.00000} ; insert
  LIN {X -7500.007,Y 2866.811,Z -169.535,A -90.84369,B 0.00000,C 180.00000} ; release
  LIN {X -7500.007,Y 2866.811,Z 130.465,A -90.84369,B 0.00000,C 180.00000} ; retreat
  ; Step 1472, bar 2026
  LIN {X -6750.007,Y 2866.811,Z 1027.751,A -90.84369,B 0.00000,C 180.00000} ; outside
  LIN {X -6750.007,Y 2866.811,Z 80.465,A -90.84369,B 0.00000,C 180.00000} ; preinsert
  LIN {X -6750.007,Y 2866.811,Z -169.535,A -90.84369,B 0.00000,C 180.00000} ; insert
  LIN {X -6750.007,Y 2866.811,Z -169.535,A -90.84369,B 0.00000,C 180.00000} ; release
  LIN {X -6750.007,Y 2866.811,Z 130.465,A -90.84369,B 0.00000,C 180.00000} ; retreat
  ; Step 1473, bar 2020
  LIN {X -6000.007,Y 2866.811,Z 1027.751,A -90.84369,B 0.00000,C 180.00000} ; outside
  LIN {X -6000.007,Y 2866.811,Z 80.465,A -90.84369,B 0.00000,C 180.00000} ; preinsert
  LIN {X -6000.007,Y 2866.811,Z -169.535,A -90.84369,B 0.00000,C 180.00000} ; insert
  LIN {X -6000.007,Y 2866.811,Z -169.535,A -90.84369,B 0.00000,C 180.00000} ; release
  LIN {X -6000.007,Y 2866.811,Z 130.465,A -90.84369,B 0.00000,C 180.00000} ; retreat
  ; Step 1474, bar 2014
  LIN {X -5250.007,Y 2866.811,Z 1027.751,A -90.84369,B 0.00000,C 180.00000} ; outside
  LIN {X -5250.007,Y 2866.811,Z 80.465,A -90.84369,B 0.00000,C 180.00000} ; preinsert
  LIN {X -5250.007,Y 2866.811,Z -169.535,A -90.84369,B 0.00000,C 180.00000} ; insert
  LIN {X -5250.007,Y 2866.811,Z -169.535,A -90.84369,B 0.00000,C 180.00000} ; release
  LIN {X -5250.007,Y 2866.811,Z 130.465,A -90.84369,B 0.00000,C 180.00000} ; retreat
  ; Step 1475, bar 2008
  LIN {X -4500.007,Y 2866.811,Z 1027.751,A -90.84369,B 0.00000,C 180.00000} ; outside
  LIN {X -4500.007,Y 2866.811,Z 80.465,A -90.84369,B 0.00000,C 180.00000} ; preinsert
  LIN {X -4500.007,Y 2866.811,Z -169.535,A -90.84369,B 0.00000,C 180.00000} ; insert
  LIN {X -4500.007,Y 2866.811,Z -169.535,A -90.84369,B 0.00000,C 180.00000} ; release
  LIN {X -4500.007,Y 2866.811,Z 130.465,A -90.84369,B 0.00000,C 180.00000} ; retreat
  ; Step 1476, bar 2002
  LIN {X -3750.007,Y 2866.811,Z 1027.751,A -90.84369,B 0.00000,C 180.00000} ; outside
  LIN {X -3750.007,Y 2866.811,Z 80.465,A -90.84369,B 0.00000,C 180.00000} ; preinsert
  LIN {X -3750.007,Y 2866.811,Z -169.535,A -90.84369,B 0.00000,C 180.00000} ; insert
  LIN {X -3750.007,Y 2866.811,Z -169.535,A -90.84369,B 0.00000,C 180.00000} ; release
  LIN {X -3750.007,Y 2866.811,Z 130.465,A -90.84369,B 0.00000,C 180.00000} ; retreat
  ; Step 1477, bar 1996
  LIN {X -3000.007,Y 2866.811,Z 1027.751,A -90.84369,B 0.00000,C 180.00000} ; outside
  LIN {X -3000.007,Y 2866.811,Z 80.465,A -90.84369,B 0.00000,C 180.00000} ; preinsert
  LIN {X -3000.007,Y 2866.811,Z -169.535,A -90.84369,B 0.00000,C 180.00000} ; insert
  LIN {X -3000.007,Y 2866.811,Z -169.535,A -90.84369,B 0.00000,C 180.00000} ; release
  LIN {X -3000.007,Y 2866.811,Z 130.465,A -90.84369,B 0.00000,C 180.00000} ; retreat
  ; Step 1478, bar 1990
  LIN {X -2250.007,Y 2866.811,Z 1027.751,A -90.84369,B 0.00000,C 180.00000} ; outside
  LIN {X -2250.007,Y 2866.811,Z 80.465,A -90.84369,B 0.00000,C 180.00000} ; preinsert
  LIN {X -2250.007,Y 2866.811,Z -169.535,A -90.84369,B 0.00000,C 180.00000} ; insert
  LIN {X -2250.007,Y 2866.811,Z -169.535,A -90.84369,B 0.00000,C 180.00000} ; release
  LIN {X -2250.007,Y 2866.811,Z 130.465,A -90.84369,B 0.00000,C 180.00000} ; retreat
  ; Step 1479, bar 1984
  LIN {X -1500.007,Y 2866.811,Z 1027.751,A -90.84369,B 0.00000,C -180.00000} ; outside
  LIN {X -1500.007,Y 2866.811,Z 80.465,A -90.84369,B 0.00000,C -180.00000} ; preinsert
  LIN {X -1500.007,Y 2866.811,Z -169.535,A -90.84369,B 0.00000,C -180.00000} ; insert
  LIN {X -1500.007,Y 2866.811,Z -169.535,A -90.84369,B 0.00000,C -180.00000} ; release
  LIN {X -1500.007,Y 2866.811,Z 130.465,A -90.84369,B 0.00000,C -180.00000} ; retreat
  ; Step 1480, bar 1978
  LIN {X -750.007,Y 2866.811,Z 1027.751,A -90.84369,B 0.00000,C -180.00000} ; outside
  LIN {X -750.007,Y 2866.811,Z 80.465,A -90.84369,B 0.00000,C -180.00000} ; preinsert
  LIN {X -750.007,Y 2866.811,Z -169.535,A -90.84369,B 0.00000,C -180.00000} ; insert
  LIN {X -750.007,Y 2866.811,Z -169.535,A -90.84369,B 0.00000,C -180.00000} ; release
  LIN {X -750.007,Y 2866.811,Z 130.465,A -90.84369,B 0.00000,C -180.00000} ; retreat
  ; Step 1481, bar 1965
  LIN {X -0.007,Y 2866.811,Z 1027.751,A -90.84369,B 0.00000,C -180.00000} ; outside
  LIN {X -0.007,Y 2866.811,Z 80.465,A -90.84369,B 0.00000,C -180.00000} ; preinsert
  LIN {X -0.007,Y 2866.811,Z -169.535,A -90.84369,B 0.00000,C -180.00000} ; insert
  LIN {X -0.007,Y 2866.811,Z -169.535,A -90.84369,B 0.00000,C -180.00000} ; release
  LIN {X -0.007,Y 2866.811,Z 130.465,A -90.84369,B 0.00000,C -180.00000} ; retreat
  ; Step 1482, bar 2116
  LIN {X 750.007,Y 2866.811,Z 1027.751,A -89.15631,B 0.00000,C 180.00000} ; outside
  LIN {X 750.007,Y 2866.811,Z 80.465,A -89.15631,B 0.00000,C 180.00000} ; preinsert
  LIN {X 750.007,Y 2866.811,Z -169.535,A -89.15631,B 0.00000,C 180.00000} ; insert
  LIN {X 750.007,Y 2866.811,Z -169.535,A -89.15631,B 0.00000,C 180.00000} ; release
  LIN {X 750.007,Y 2866.811,Z 130.465,A -89.15631,B 0.00000,C 180.00000} ; retreat
  ; Step 1483, bar 2122
  LIN {X 1500.007,Y 2866.811,Z 1027.751,A -89.15631,B 0.00000,C -180.00000} ; outside
  LIN {X 1500.007,Y 2866.811,Z 80.465,A -89.15631,B 0.00000,C -180.00000} ; preinsert
  LIN {X 1500.007,Y 2866.811,Z -169.535,A -89.15631,B 0.00000,C -180.00000} ; insert
  LIN {X 1500.007,Y 2866.811,Z -169.535,A -89.15631,B 0.00000,C -180.00000} ; release
  LIN {X 1500.007,Y 2866.811,Z 130.465,A -89.15631,B 0.00000,C -180.00000} ; retreat
  ; Step 1484, bar 2128
  LIN {X 2250.007,Y 2866.811,Z 1027.751,A -89.15631,B 0.00000,C 180.00000} ; outside
  LIN {X 2250.007,Y 2866.811,Z 80.465,A -89.15631,B 0.00000,C 180.00000} ; preinsert
  LIN {X 2250.007,Y 2866.811,Z -169.535,A -89.15631,B 0.00000,C 180.00000} ; insert
  LIN {X 2250.007,Y 2866.811,Z -169.535,A -89.15631,B 0.00000,C 180.00000} ; release
  LIN {X 2250.007,Y 2866.811,Z 130.465,A -89.15631,B 0.00000,C 180.00000} ; retreat
  ; Step 1485, bar 2134
  LIN {X 3000.007,Y 2866.811,Z 1027.751,A -89.15631,B 0.00000,C 180.00000} ; outside
  LIN {X 3000.007,Y 2866.811,Z 80.465,A -89.15631,B 0.00000,C 180.00000} ; preinsert
  LIN {X 3000.007,Y 2866.811,Z -169.535,A -89.15631,B 0.00000,C 180.00000} ; insert
  LIN {X 3000.007,Y 2866.811,Z -169.535,A -89.15631,B 0.00000,C 180.00000} ; release
  LIN {X 3000.007,Y 2866.811,Z 130.465,A -89.15631,B 0.00000,C 180.00000} ; retreat
  ; Step 1486, bar 2140
  LIN {X 3750.007,Y 2866.811,Z 1027.751,A -89.15631,B 0.00000,C 180.00000} ; outside
  LIN {X 3750.007,Y 2866.811,Z 80.465,A -89.15631,B 0.00000,C 180.00000} ; preinsert
  LIN {X 3750.007,Y 2866.811,Z -169.535,A -89.15631,B 0.00000,C 180.00000} ; insert
  LIN {X 3750.007,Y 2866.811,Z -169.535,A -89.15631,B 0.00000,C 180.00000} ; release
  LIN {X 3750.007,Y 2866.811,Z 130.465,A -89.15631,B 0.00000,C 180.00000} ; retreat
  ; Step 1487, bar 2146
  LIN {X 4500.007,Y 2866.811,Z 1027.751,A -89.15631,B 0.00000,C 180.00000} ; outside
  LIN {X 4500.007,Y 2866.811,Z 80.465,A -89.15631,B 0.00000,C 180.00000} ; preinsert
  LIN {X 4500.007,Y 2866.811,Z -169.535,A -89.15631,B 0.00000,C 180.00000} ; insert
  LIN {X 4500.007,Y 2866.811,Z -169.535,A -89.15631,B 0.00000,C 180.00000} ; release
  LIN {X 4500.007,Y 2866.811,Z 130.465,A -89.15631,B 0.00000,C 180.00000} ; retreat
  ; Step 1488, bar 2152
  LIN {X 5250.007,Y 2866.811,Z 1027.751,A -89.15631,B 0.00000,C 180.00000} ; outside
  LIN {X 5250.007,Y 2866.811,Z 80.465,A -89.15631,B 0.00000,C 180.00000} ; preinsert
  LIN {X 5250.007,Y 2866.811,Z -169.535,A -89.15631,B 0.00000,C 180.00000} ; insert
  LIN {X 5250.007,Y 2866.811,Z -169.535,A -89.15631,B 0.00000,C 180.00000} ; release
  LIN {X 5250.007,Y 2866.811,Z 130.465,A -89.15631,B 0.00000,C 180.00000} ; retreat
  ; Step 1489, bar 2158
  LIN {X 6000.007,Y 2866.811,Z 1027.751,A -89.15631,B 0.00000,C 180.00000} ; outside
  LIN {X 6000.007,Y 2866.811,Z 80.465,A -89.15631,B 0.00000,C 180.00000} ; preinsert
  LIN {X 6000.007,Y 2866.811,Z -169.535,A -89.15631,B 0.00000,C 180.00000} ; insert
  LIN {X 6000.007,Y 2866.811,Z -169.535,A -89.15631,B 0.00000,C 180.00000} ; release
  LIN {X 6000.007,Y 2866.811,Z 130.465,A -89.15631,B 0.00000,C 180.00000} ; retreat
  ; Step 1490, bar 2164
  LIN {X 6750.007,Y 2866.811,Z 1027.751,A -89.15631,B 0.00000,C 180.00000} ; outside
  LIN {X 6750.007,Y 2866.811,Z 80.465,A -89.15631,B 0.00000,C 180.00000} ; preinsert
  LIN {X 6750.007,Y 2866.811,Z -169.535,A -89.15631,B 0.00000,C 180.00000} ; insert
  LIN {X 6750.007,Y 2866.811,Z -169.535,A -89.15631,B 0.00000,C 180.00000} ; release
  LIN {X 6750.007,Y 2866.811,Z 130.465,A -89.15631,B 0.00000,C 180.00000} ; retreat
  ; Step 1491, bar 2170
  LIN {X 7500.007,Y 2866.811,Z 1027.751,A -89.15631,B 0.00000,C 180.00000} ; outside
  LIN {X 7500.007,Y 2866.811,Z 80.465,A -89.15631,B 0.00000,C 180.00000} ; preinsert
  LIN {X 7500.007,Y 2866.811,Z -169.535,A -89.15631,B 0.00000,C 180.00000} ; insert
  LIN {X 7500.007,Y 2866.811,Z -169.535,A -89.15631,B 0.00000,C 180.00000} ; release
  LIN {X 7500.007,Y 2866.811,Z 130.465,A -89.15631,B 0.00000,C 180.00000} ; retreat
  ; Step 1492, bar 2176
  LIN {X 8250.007,Y 2866.811,Z 1027.751,A -89.15631,B 0.00000,C 180.00000} ; outside
  LIN {X 8250.007,Y 2866.811,Z 80.465,A -89.15631,B 0.00000,C 180.00000} ; preinsert
  LIN {X 8250.007,Y 2866.811,Z -169.535,A -89.15631,B 0.00000,C 180.00000} ; insert
  LIN {X 8250.007,Y 2866.811,Z -169.535,A -89.15631,B 0.00000,C 180.00000} ; release
  LIN {X 8250.007,Y 2866.811,Z 130.465,A -89.15631,B 0.00000,C 180.00000} ; retreat
  ; Step 1493, bar 2182
  LIN {X 9000.007,Y 2866.811,Z 1027.751,A -89.15631,B 0.00000,C 180.00000} ; outside
  LIN {X 9000.007,Y 2866.811,Z 80.465,A -89.15631,B 0.00000,C 180.00000} ; preinsert
  LIN {X 9000.007,Y 2866.811,Z -169.535,A -89.15631,B 0.00000,C 180.00000} ; insert
  LIN {X 9000.007,Y 2866.811,Z -169.535,A -89.15631,B 0.00000,C 180.00000} ; release
  LIN {X 9000.007,Y 2866.811,Z 130.465,A -89.15631,B 0.00000,C 180.00000} ; retreat
  ; Step 1494, bar 2188
  LIN {X 9750.007,Y 2866.811,Z 1027.751,A -89.15631,B 0.00000,C 180.00000} ; outside
  LIN {X 9750.007,Y 2866.811,Z 80.465,A -89.15631,B 0.00000,C 180.00000} ; preinsert
  LIN {X 9750.007,Y 2866.811,Z -169.535,A -89.15631,B 0.00000,C 180.00000} ; insert
  LIN {X 9750.007,Y 2866.811,Z -169.535,A -89.15631,B 0.00000,C 180.00000} ; release
  LIN {X 9750.007,Y 2866.811,Z 130.465,A -89.15631,B 0.00000,C 180.00000} ; retreat
  ; Step 1495, bar 2194
  LIN {X 10500.007,Y 2866.811,Z 1027.751,A -89.15631,B 0.00000,C 180.00000} ; outside
  LIN {X 10500.007,Y 2866.811,Z 80.465,A -89.15631,B 0.00000,C 180.00000} ; preinsert
  LIN {X 10500.007,Y 2866.811,Z -169.535,A -89.15631,B 0.00000,C 180.00000} ; insert
  LIN {X 10500.007,Y 2866.811,Z -169.535,A -89.15631,B 0.00000,C 180.00000} ; release
  LIN {X 10500.007,Y 2866.811,Z 130.465,A -89.15631,B 0.00000,C 180.00000} ; retreat
  ; Step 1496, bar 2200
  LIN {X 11250.007,Y 2866.811,Z 1027.751,A -89.15631,B 0.00000,C 180.00000} ; outside
  LIN {X 11250.007,Y 2866.811,Z 80.465,A -89.15631,B 0.00000,C 180.00000} ; preinsert
  LIN {X 11250.007,Y 2866.811,Z -169.535,A -89.15631,B 0.00000,C 180.00000} ; insert
  LIN {X 11250.007,Y 2866.811,Z -169.535,A -89.15631,B 0.00000,C 180.00000} ; release
  LIN {X 11250.007,Y 2866.811,Z 130.465,A -89.15631,B 0.00000,C 180.00000} ; retreat
  ; Step 1497, bar 2206
  LIN {X 12000.007,Y 2866.811,Z 1027.751,A -89.15631,B 0.00000,C 180.00000} ; outside
  LIN {X 12000.007,Y 2866.811,Z 80.465,A -89.15631,B 0.00000,C 180.00000} ; preinsert
  LIN {X 12000.007,Y 2866.811,Z -169.535,A -89.15631,B 0.00000,C 180.00000} ; insert
  LIN {X 12000.007,Y 2866.811,Z -169.535,A -89.15631,B 0.00000,C 180.00000} ; release
  LIN {X 12000.007,Y 2866.811,Z 130.465,A -89.15631,B 0.00000,C 180.00000} ; retreat
  ; Step 1498, bar 2211
  LIN {X 12550.007,Y 2866.811,Z 1027.751,A -89.15631,B 0.00000,C 180.00000} ; outside
  LIN {X 12550.007,Y 2866.811,Z 80.465,A -89.15631,B 0.00000,C 180.00000} ; preinsert
  LIN {X 12550.007,Y 2866.811,Z -169.535,A -89.15631,B 0.00000,C 180.00000} ; insert
  LIN {X 12550.007,Y 2866.811,Z -169.535,A -89.15631,B 0.00000,C 180.00000} ; release
  LIN {X 12550.007,Y 2866.811,Z 130.465,A -89.15631,B 0.00000,C 180.00000} ; retreat
  ; Step 1499, bar 2217
  LIN {X 13150.007,Y 2866.811,Z 1027.751,A -89.15631,B 0.00000,C 180.00000} ; outside
  LIN {X 13150.007,Y 2866.811,Z 80.465,A -89.15631,B 0.00000,C 180.00000} ; preinsert
  LIN {X 13150.007,Y 2866.811,Z -169.535,A -89.15631,B 0.00000,C 180.00000} ; insert
  LIN {X 13150.007,Y 2866.811,Z -169.535,A -89.15631,B 0.00000,C 180.00000} ; release
  LIN {X 13150.007,Y 2866.811,Z 130.465,A -89.15631,B 0.00000,C 180.00000} ; retreat
  ; Step 1500, bar 2223
  LIN {X 13750.007,Y 2866.811,Z 1027.751,A -89.15631,B 0.00000,C 180.00000} ; outside
  LIN {X 13750.007,Y 2866.811,Z 80.465,A -89.15631,B 0.00000,C 180.00000} ; preinsert
  LIN {X 13750.007,Y 2866.811,Z -169.535,A -89.15631,B 0.00000,C 180.00000} ; insert
  LIN {X 13750.007,Y 2866.811,Z -169.535,A -89.15631,B 0.00000,C 180.00000} ; release
  LIN {X 13750.007,Y 2866.811,Z 130.465,A -89.15631,B 0.00000,C 180.00000} ; retreat
  ; Step 1501, bar 2229
  LIN {X 14350.007,Y 2866.811,Z 1027.751,A -89.15631,B 0.00000,C 180.00000} ; outside
  LIN {X 14350.007,Y 2866.811,Z 80.465,A -89.15631,B 0.00000,C 180.00000} ; preinsert
  LIN {X 14350.007,Y 2866.811,Z -169.535,A -89.15631,B 0.00000,C 180.00000} ; insert
  LIN {X 14350.007,Y 2866.811,Z -169.535,A -89.15631,B 0.00000,C 180.00000} ; release
  LIN {X 14350.007,Y 2866.811,Z 130.465,A -89.15631,B 0.00000,C 180.00000} ; retreat
  ; Step 1502, bar 2235
  LIN {X 14950.007,Y 2866.811,Z 1027.751,A -89.15631,B 0.00000,C 180.00000} ; outside
  LIN {X 14950.007,Y 2866.811,Z 80.465,A -89.15631,B 0.00000,C 180.00000} ; preinsert
  LIN {X 14950.007,Y 2866.811,Z -169.535,A -89.15631,B 0.00000,C 180.00000} ; insert
  LIN {X 14950.007,Y 2866.811,Z -169.535,A -89.15631,B 0.00000,C 180.00000} ; release
  LIN {X 14950.007,Y 2866.811,Z 130.465,A -89.15631,B 0.00000,C 180.00000} ; retreat
  ; Step 1503, bar 2241
  LIN {X 15550.007,Y 2866.811,Z 1027.751,A -89.15631,B 0.00000,C 180.00000} ; outside
  LIN {X 15550.007,Y 2866.811,Z 80.465,A -89.15631,B 0.00000,C 180.00000} ; preinsert
  LIN {X 15550.007,Y 2866.811,Z -169.535,A -89.15631,B 0.00000,C 180.00000} ; insert
  LIN {X 15550.007,Y 2866.811,Z -169.535,A -89.15631,B 0.00000,C 180.00000} ; release
  LIN {X 15550.007,Y 2866.811,Z 130.465,A -89.15631,B 0.00000,C 180.00000} ; retreat
  ; Step 1504, bar 2247
  LIN {X 16150.007,Y 2866.811,Z 1027.751,A -89.15631,B 0.00000,C 180.00000} ; outside
  LIN {X 16150.007,Y 2866.811,Z 80.465,A -89.15631,B 0.00000,C 180.00000} ; preinsert
  LIN {X 16150.007,Y 2866.811,Z -169.535,A -89.15631,B 0.00000,C 180.00000} ; insert
  LIN {X 16150.007,Y 2866.811,Z -169.535,A -89.15631,B 0.00000,C 180.00000} ; release
  LIN {X 16150.007,Y 2866.811,Z 130.465,A -89.15631,B 0.00000,C 180.00000} ; retreat
  ; Step 1505, bar 3050
  LIN {X -16049.996,Y -1026.029,Z 973.273,A -172.46345,B 0.00000,C -180.00000} ; outside
  LIN {X -16049.996,Y -1026.029,Z 17.643,A -172.46345,B 0.00000,C -180.00000} ; preinsert
  LIN {X -16049.996,Y -1026.029,Z -232.357,A -172.46345,B 0.00000,C -180.00000} ; insert
  LIN {X -16049.996,Y -1026.029,Z -232.357,A -172.46345,B 0.00000,C -180.00000} ; release
  LIN {X -16049.996,Y -1026.029,Z 67.643,A -172.46345,B 0.00000,C -180.00000} ; retreat
  ; Step 1506, bar 3045
  LIN {X -15649.996,Y -1026.029,Z 973.273,A -172.46345,B 0.00000,C -180.00000} ; outside
  LIN {X -15649.996,Y -1026.029,Z 17.643,A -172.46345,B 0.00000,C -180.00000} ; preinsert
  LIN {X -15649.996,Y -1026.029,Z -232.357,A -172.46345,B 0.00000,C -180.00000} ; insert
  LIN {X -15649.996,Y -1026.029,Z -232.357,A -172.46345,B 0.00000,C -180.00000} ; release
  LIN {X -15649.996,Y -1026.029,Z 67.643,A -172.46345,B 0.00000,C -180.00000} ; retreat
  ; Step 1507, bar 3040
  LIN {X -15249.996,Y -1026.029,Z 973.273,A -172.46345,B 0.00000,C -180.00000} ; outside
  LIN {X -15249.996,Y -1026.029,Z 17.643,A -172.46345,B 0.00000,C -180.00000} ; preinsert
  LIN {X -15249.996,Y -1026.029,Z -232.357,A -172.46345,B 0.00000,C -180.00000} ; insert
  LIN {X -15249.996,Y -1026.029,Z -232.357,A -172.46345,B 0.00000,C -180.00000} ; release
  LIN {X -15249.996,Y -1026.029,Z 67.643,A -172.46345,B 0.00000,C -180.00000} ; retreat
  ; Step 1508, bar 3055
  LIN {X 15249.996,Y 1026.029,Z 973.273,A 7.53655,B 0.00000,C 180.00000} ; outside
  LIN {X 15249.996,Y 1026.029,Z 17.643,A 7.53655,B 0.00000,C 180.00000} ; preinsert
  LIN {X 15249.996,Y 1026.029,Z -232.357,A 7.53655,B 0.00000,C 180.00000} ; insert
  LIN {X 15249.996,Y 1026.029,Z -232.357,A 7.53655,B 0.00000,C 180.00000} ; release
  LIN {X 15249.996,Y 1026.029,Z 67.643,A 7.53655,B 0.00000,C 180.00000} ; retreat
  ; Step 1509, bar 3061
  LIN {X 15649.996,Y 1026.029,Z 973.273,A 7.53655,B 0.00000,C 180.00000} ; outside
  LIN {X 15649.996,Y 1026.029,Z 17.643,A 7.53655,B 0.00000,C 180.00000} ; preinsert
  LIN {X 15649.996,Y 1026.029,Z -232.357,A 7.53655,B 0.00000,C 180.00000} ; insert
  LIN {X 15649.996,Y 1026.029,Z -232.357,A 7.53655,B 0.00000,C 180.00000} ; release
  LIN {X 15649.996,Y 1026.029,Z 67.643,A 7.53655,B 0.00000,C 180.00000} ; retreat
  ; Step 1510, bar 3067
  LIN {X 16049.996,Y 1026.029,Z 973.273,A 7.53655,B 0.00000,C 180.00000} ; outside
  LIN {X 16049.996,Y 1026.029,Z 17.643,A 7.53655,B 0.00000,C 180.00000} ; preinsert
  LIN {X 16049.996,Y 1026.029,Z -232.357,A 7.53655,B 0.00000,C 180.00000} ; insert
  LIN {X 16049.996,Y 1026.029,Z -232.357,A 7.53655,B 0.00000,C 180.00000} ; release
  LIN {X 16049.996,Y 1026.029,Z 67.643,A 7.53655,B 0.00000,C 180.00000} ; retreat
  ; Step 1511, bar 3073
  LIN {X 15249.996,Y -1026.029,Z 973.274,A -7.53655,B 0.00000,C 180.00000} ; outside
  LIN {X 15249.996,Y -1026.029,Z 17.643,A -7.53655,B 0.00000,C 180.00000} ; preinsert
  LIN {X 15249.996,Y -1026.029,Z -232.357,A -7.53655,B 0.00000,C 180.00000} ; insert
  LIN {X 15249.996,Y -1026.029,Z -232.357,A -7.53655,B 0.00000,C 180.00000} ; release
  LIN {X 15249.996,Y -1026.029,Z 67.643,A -7.53655,B 0.00000,C 180.00000} ; retreat
  ; Step 1512, bar 3078
  LIN {X 15649.996,Y -1026.029,Z 973.274,A -7.53655,B 0.00000,C 180.00000} ; outside
  LIN {X 15649.996,Y -1026.029,Z 17.643,A -7.53655,B 0.00000,C 180.00000} ; preinsert
  LIN {X 15649.996,Y -1026.029,Z -232.357,A -7.53655,B 0.00000,C 180.00000} ; insert
  LIN {X 15649.996,Y -1026.029,Z -232.357,A -7.53655,B 0.00000,C 180.00000} ; release
  LIN {X 15649.996,Y -1026.029,Z 67.643,A -7.53655,B 0.00000,C 180.00000} ; retreat
  ; Step 1513, bar 3083
  LIN {X 16049.996,Y -1026.029,Z 973.274,A -7.53655,B 0.00000,C 180.00000} ; outside
  LIN {X 16049.996,Y -1026.029,Z 17.643,A -7.53655,B 0.00000,C 180.00000} ; preinsert
  LIN {X 16049.996,Y -1026.029,Z -232.357,A -7.53655,B 0.00000,C 180.00000} ; insert
  LIN {X 16049.996,Y -1026.029,Z -232.357,A -7.53655,B 0.00000,C 180.00000} ; release
  LIN {X 16049.996,Y -1026.029,Z 67.643,A -7.53655,B 0.00000,C 180.00000} ; retreat
  ; Step 1514, bar 3034
  LIN {X -16049.996,Y 1026.029,Z 973.274,A 172.46345,B 0.00000,C 180.00000} ; outside
  LIN {X -16049.996,Y 1026.029,Z 17.643,A 172.46345,B 0.00000,C 180.00000} ; preinsert
  LIN {X -16049.996,Y 1026.029,Z -232.357,A 172.46345,B 0.00000,C 180.00000} ; insert
  LIN {X -16049.996,Y 1026.029,Z -232.357,A 172.46345,B 0.00000,C 180.00000} ; release
  LIN {X -16049.996,Y 1026.029,Z 67.643,A 172.46345,B 0.00000,C 180.00000} ; retreat
  ; Step 1515, bar 3028
  LIN {X -15649.996,Y 1026.029,Z 973.274,A 172.46345,B 0.00000,C 180.00000} ; outside
  LIN {X -15649.996,Y 1026.029,Z 17.643,A 172.46345,B 0.00000,C 180.00000} ; preinsert
  LIN {X -15649.996,Y 1026.029,Z -232.357,A 172.46345,B 0.00000,C 180.00000} ; insert
  LIN {X -15649.996,Y 1026.029,Z -232.357,A 172.46345,B 0.00000,C 180.00000} ; release
  LIN {X -15649.996,Y 1026.029,Z 67.643,A 172.46345,B 0.00000,C 180.00000} ; retreat
  ; Step 1516, bar 3022
  LIN {X -15249.996,Y 1026.029,Z 973.274,A 172.46345,B 0.00000,C 180.00000} ; outside
  LIN {X -15249.996,Y 1026.029,Z 17.643,A 172.46345,B 0.00000,C 180.00000} ; preinsert
  LIN {X -15249.996,Y 1026.029,Z -232.357,A 172.46345,B 0.00000,C 180.00000} ; insert
  LIN {X -15249.996,Y 1026.029,Z -232.357,A 172.46345,B 0.00000,C 180.00000} ; release
  LIN {X -15249.996,Y 1026.029,Z 67.643,A 172.46345,B 0.00000,C 180.00000} ; retreat
  ; Step 1517, bar 2522
  LIN {X 15849.916,Y -3131.796,Z 1047.576,A 92.55766,B 0.00000,C -180.00000} ; outside
  LIN {X 15849.916,Y -3131.796,Z 96.905,A 92.55766,B 0.00000,C -180.00000} ; preinsert
  LIN {X 15849.916,Y -3131.796,Z -153.095,A 92.55766,B 0.00000,C -180.00000} ; insert
  LIN {X 15849.916,Y -3131.796,Z -153.095,A 92.55766,B 0.00000,C -180.00000} ; release
  LIN {X 15849.916,Y -3131.796,Z 146.905,A 92.55766,B 0.00000,C -180.00000} ; retreat
  ; Step 1518, bar 2516
  LIN {X 15249.916,Y -3131.796,Z 1047.576,A 92.55766,B 0.00000,C -180.00000} ; outside
  LIN {X 15249.916,Y -3131.796,Z 96.905,A 92.55766,B 0.00000,C -180.00000} ; preinsert
  LIN {X 15249.916,Y -3131.796,Z -153.095,A 92.55766,B 0.00000,C -180.00000} ; insert
  LIN {X 15249.916,Y -3131.796,Z -153.095,A 92.55766,B 0.00000,C -180.00000} ; release
  LIN {X 15249.916,Y -3131.796,Z 146.905,A 92.55766,B 0.00000,C -180.00000} ; retreat
  ; Step 1519, bar 2510
  LIN {X 14649.916,Y -3131.796,Z 1047.576,A 92.55766,B 0.00000,C -180.00000} ; outside
  LIN {X 14649.916,Y -3131.796,Z 96.905,A 92.55766,B 0.00000,C -180.00000} ; preinsert
  LIN {X 14649.916,Y -3131.796,Z -153.095,A 92.55766,B 0.00000,C -180.00000} ; insert
  LIN {X 14649.916,Y -3131.796,Z -153.095,A 92.55766,B 0.00000,C -180.00000} ; release
  LIN {X 14649.916,Y -3131.796,Z 146.905,A 92.55766,B 0.00000,C -180.00000} ; retreat
  ; Step 1520, bar 2504
  LIN {X 14049.916,Y -3131.796,Z 1047.576,A 92.55766,B 0.00000,C -180.00000} ; outside
  LIN {X 14049.916,Y -3131.796,Z 96.905,A 92.55766,B 0.00000,C -180.00000} ; preinsert
  LIN {X 14049.916,Y -3131.796,Z -153.095,A 92.55766,B 0.00000,C -180.00000} ; insert
  LIN {X 14049.916,Y -3131.796,Z -153.095,A 92.55766,B 0.00000,C -180.00000} ; release
  LIN {X 14049.916,Y -3131.796,Z 146.905,A 92.55766,B 0.00000,C -180.00000} ; retreat
  ; Step 1521, bar 2498
  LIN {X 13449.916,Y -3131.796,Z 1047.576,A 92.55766,B 0.00000,C -180.00000} ; outside
  LIN {X 13449.916,Y -3131.796,Z 96.905,A 92.55766,B 0.00000,C -180.00000} ; preinsert
  LIN {X 13449.916,Y -3131.796,Z -153.095,A 92.55766,B 0.00000,C -180.00000} ; insert
  LIN {X 13449.916,Y -3131.796,Z -153.095,A 92.55766,B 0.00000,C -180.00000} ; release
  LIN {X 13449.916,Y -3131.796,Z 146.905,A 92.55766,B 0.00000,C -180.00000} ; retreat
  ; Step 1522, bar 2492
  LIN {X 12849.916,Y -3131.796,Z 1047.576,A 92.55766,B 0.00000,C -180.00000} ; outside
  LIN {X 12849.916,Y -3131.796,Z 96.905,A 92.55766,B 0.00000,C -180.00000} ; preinsert
  LIN {X 12849.916,Y -3131.796,Z -153.095,A 92.55766,B 0.00000,C -180.00000} ; insert
  LIN {X 12849.916,Y -3131.796,Z -153.095,A 92.55766,B 0.00000,C -180.00000} ; release
  LIN {X 12849.916,Y -3131.796,Z 146.905,A 92.55766,B 0.00000,C -180.00000} ; retreat
  ; Step 1523, bar 2484
  LIN {X 12249.916,Y -3131.796,Z 1047.576,A 92.55766,B 0.00000,C -180.00000} ; outside
  LIN {X 12249.916,Y -3131.796,Z 96.905,A 92.55766,B 0.00000,C -180.00000} ; preinsert
  LIN {X 12249.916,Y -3131.796,Z -153.095,A 92.55766,B 0.00000,C -180.00000} ; insert
  LIN {X 12249.916,Y -3131.796,Z -153.095,A 92.55766,B 0.00000,C -180.00000} ; release
  LIN {X 12249.916,Y -3131.796,Z 146.905,A 92.55766,B 0.00000,C -180.00000} ; retreat
  ; Step 1524, bar 2478
  LIN {X 11624.916,Y -3131.796,Z 1047.576,A 92.55766,B 0.00000,C -180.00000} ; outside
  LIN {X 11624.916,Y -3131.796,Z 96.905,A 92.55766,B 0.00000,C -180.00000} ; preinsert
  LIN {X 11624.916,Y -3131.796,Z -153.095,A 92.55766,B 0.00000,C -180.00000} ; insert
  LIN {X 11624.916,Y -3131.796,Z -153.095,A 92.55766,B 0.00000,C -180.00000} ; release
  LIN {X 11624.916,Y -3131.796,Z 146.905,A 92.55766,B 0.00000,C -180.00000} ; retreat
  ; Step 1525, bar 2472
  LIN {X 10874.916,Y -3131.796,Z 1047.576,A 92.55766,B 0.00000,C -180.00000} ; outside
  LIN {X 10874.916,Y -3131.796,Z 96.905,A 92.55766,B 0.00000,C -180.00000} ; preinsert
  LIN {X 10874.916,Y -3131.796,Z -153.095,A 92.55766,B 0.00000,C -180.00000} ; insert
  LIN {X 10874.916,Y -3131.796,Z -153.095,A 92.55766,B 0.00000,C -180.00000} ; release
  LIN {X 10874.916,Y -3131.796,Z 146.905,A 92.55766,B 0.00000,C -180.00000} ; retreat
  ; Step 1526, bar 2466
  LIN {X 10124.916,Y -3131.796,Z 1047.576,A 92.55766,B 0.00000,C -180.00000} ; outside
  LIN {X 10124.916,Y -3131.796,Z 96.905,A 92.55766,B 0.00000,C -180.00000} ; preinsert
  LIN {X 10124.916,Y -3131.796,Z -153.095,A 92.55766,B 0.00000,C -180.00000} ; insert
  LIN {X 10124.916,Y -3131.796,Z -153.095,A 92.55766,B 0.00000,C -180.00000} ; release
  LIN {X 10124.916,Y -3131.796,Z 146.905,A 92.55766,B 0.00000,C -180.00000} ; retreat
  ; Step 1527, bar 2460
  LIN {X 9374.916,Y -3131.796,Z 1047.576,A 92.55766,B 0.00000,C -180.00000} ; outside
  LIN {X 9374.916,Y -3131.796,Z 96.905,A 92.55766,B 0.00000,C -180.00000} ; preinsert
  LIN {X 9374.916,Y -3131.796,Z -153.095,A 92.55766,B 0.00000,C -180.00000} ; insert
  LIN {X 9374.916,Y -3131.796,Z -153.095,A 92.55766,B 0.00000,C -180.00000} ; release
  LIN {X 9374.916,Y -3131.796,Z 146.905,A 92.55766,B 0.00000,C -180.00000} ; retreat
  ; Step 1528, bar 2454
  LIN {X 8624.916,Y -3131.796,Z 1047.576,A 92.55766,B 0.00000,C -180.00000} ; outside
  LIN {X 8624.916,Y -3131.796,Z 96.905,A 92.55766,B 0.00000,C -180.00000} ; preinsert
  LIN {X 8624.916,Y -3131.796,Z -153.095,A 92.55766,B 0.00000,C -180.00000} ; insert
  LIN {X 8624.916,Y -3131.796,Z -153.095,A 92.55766,B 0.00000,C -180.00000} ; release
  LIN {X 8624.916,Y -3131.796,Z 146.905,A 92.55766,B 0.00000,C -180.00000} ; retreat
  ; Step 1529, bar 2448
  LIN {X 7874.916,Y -3131.796,Z 1047.576,A 92.55766,B 0.00000,C 180.00000} ; outside
  LIN {X 7874.916,Y -3131.796,Z 96.905,A 92.55766,B 0.00000,C 180.00000} ; preinsert
  LIN {X 7874.916,Y -3131.796,Z -153.095,A 92.55766,B 0.00000,C 180.00000} ; insert
  LIN {X 7874.916,Y -3131.796,Z -153.095,A 92.55766,B 0.00000,C 180.00000} ; release
  LIN {X 7874.916,Y -3131.796,Z 146.905,A 92.55766,B 0.00000,C 180.00000} ; retreat
  ; Step 1530, bar 2442
  LIN {X 7124.916,Y -3131.796,Z 1047.576,A 92.55766,B 0.00000,C 180.00000} ; outside
  LIN {X 7124.916,Y -3131.796,Z 96.905,A 92.55766,B 0.00000,C 180.00000} ; preinsert
  LIN {X 7124.916,Y -3131.796,Z -153.095,A 92.55766,B 0.00000,C 180.00000} ; insert
  LIN {X 7124.916,Y -3131.796,Z -153.095,A 92.55766,B 0.00000,C 180.00000} ; release
  LIN {X 7124.916,Y -3131.796,Z 146.905,A 92.55766,B 0.00000,C 180.00000} ; retreat
  ; Step 1531, bar 2436
  LIN {X 6374.916,Y -3131.796,Z 1047.576,A 92.55766,B 0.00000,C 180.00000} ; outside
  LIN {X 6374.916,Y -3131.796,Z 96.905,A 92.55766,B 0.00000,C 180.00000} ; preinsert
  LIN {X 6374.916,Y -3131.796,Z -153.095,A 92.55766,B 0.00000,C 180.00000} ; insert
  LIN {X 6374.916,Y -3131.796,Z -153.095,A 92.55766,B 0.00000,C 180.00000} ; release
  LIN {X 6374.916,Y -3131.796,Z 146.905,A 92.55766,B 0.00000,C 180.00000} ; retreat
  ; Step 1532, bar 2430
  LIN {X 5624.916,Y -3131.796,Z 1047.576,A 92.55766,B 0.00000,C 180.00000} ; outside
  LIN {X 5624.916,Y -3131.796,Z 96.905,A 92.55766,B 0.00000,C 180.00000} ; preinsert
  LIN {X 5624.916,Y -3131.796,Z -153.095,A 92.55766,B 0.00000,C 180.00000} ; insert
  LIN {X 5624.916,Y -3131.796,Z -153.095,A 92.55766,B 0.00000,C 180.00000} ; release
  LIN {X 5624.916,Y -3131.796,Z 146.905,A 92.55766,B 0.00000,C 180.00000} ; retreat
  ; Step 1533, bar 2424
  LIN {X 4874.916,Y -3131.796,Z 1047.576,A 92.55766,B 0.00000,C 180.00000} ; outside
  LIN {X 4874.916,Y -3131.796,Z 96.905,A 92.55766,B 0.00000,C 180.00000} ; preinsert
  LIN {X 4874.916,Y -3131.796,Z -153.095,A 92.55766,B 0.00000,C 180.00000} ; insert
  LIN {X 4874.916,Y -3131.796,Z -153.095,A 92.55766,B 0.00000,C 180.00000} ; release
  LIN {X 4874.916,Y -3131.796,Z 146.905,A 92.55766,B 0.00000,C 180.00000} ; retreat
  ; Step 1534, bar 2418
  LIN {X 4124.916,Y -3131.796,Z 1047.576,A 92.55766,B 0.00000,C 180.00000} ; outside
  LIN {X 4124.916,Y -3131.796,Z 96.905,A 92.55766,B 0.00000,C 180.00000} ; preinsert
  LIN {X 4124.916,Y -3131.796,Z -153.095,A 92.55766,B 0.00000,C 180.00000} ; insert
  LIN {X 4124.916,Y -3131.796,Z -153.095,A 92.55766,B 0.00000,C 180.00000} ; release
  LIN {X 4124.916,Y -3131.796,Z 146.905,A 92.55766,B 0.00000,C 180.00000} ; retreat
  ; Step 1535, bar 2412
  LIN {X 3374.916,Y -3131.796,Z 1047.576,A 92.55766,B 0.00000,C -180.00000} ; outside
  LIN {X 3374.916,Y -3131.796,Z 96.905,A 92.55766,B 0.00000,C -180.00000} ; preinsert
  LIN {X 3374.916,Y -3131.796,Z -153.095,A 92.55766,B 0.00000,C -180.00000} ; insert
  LIN {X 3374.916,Y -3131.796,Z -153.095,A 92.55766,B 0.00000,C -180.00000} ; release
  LIN {X 3374.916,Y -3131.796,Z 146.905,A 92.55766,B 0.00000,C -180.00000} ; retreat
  ; Step 1536, bar 2406
  LIN {X 2624.916,Y -3131.796,Z 1047.576,A 92.55766,B 0.00000,C -180.00000} ; outside
  LIN {X 2624.916,Y -3131.796,Z 96.905,A 92.55766,B 0.00000,C -180.00000} ; preinsert
  LIN {X 2624.916,Y -3131.796,Z -153.095,A 92.55766,B 0.00000,C -180.00000} ; insert
  LIN {X 2624.916,Y -3131.796,Z -153.095,A 92.55766,B 0.00000,C -180.00000} ; release
  LIN {X 2624.916,Y -3131.796,Z 146.905,A 92.55766,B 0.00000,C -180.00000} ; retreat
  ; Step 1537, bar 2400
  LIN {X 1874.916,Y -3131.796,Z 1047.576,A 92.55766,B 0.00000,C 180.00000} ; outside
  LIN {X 1874.916,Y -3131.796,Z 96.905,A 92.55766,B 0.00000,C 180.00000} ; preinsert
  LIN {X 1874.916,Y -3131.796,Z -153.095,A 92.55766,B 0.00000,C 180.00000} ; insert
  LIN {X 1874.916,Y -3131.796,Z -153.095,A 92.55766,B 0.00000,C 180.00000} ; release
  LIN {X 1874.916,Y -3131.796,Z 146.905,A 92.55766,B 0.00000,C 180.00000} ; retreat
  ; Step 1538, bar 2394
  LIN {X 1124.916,Y -3131.796,Z 1047.576,A 92.55766,B 0.00000,C 180.00000} ; outside
  LIN {X 1124.916,Y -3131.796,Z 96.905,A 92.55766,B 0.00000,C 180.00000} ; preinsert
  LIN {X 1124.916,Y -3131.796,Z -153.095,A 92.55766,B 0.00000,C 180.00000} ; insert
  LIN {X 1124.916,Y -3131.796,Z -153.095,A 92.55766,B 0.00000,C 180.00000} ; release
  LIN {X 1124.916,Y -3131.796,Z 146.905,A 92.55766,B 0.00000,C 180.00000} ; retreat
  ; Step 1539, bar 2390
  LIN {X 374.916,Y -3131.796,Z 1047.576,A 92.55766,B 0.00000,C -180.00000} ; outside
  LIN {X 374.916,Y -3131.796,Z 96.905,A 92.55766,B 0.00000,C -180.00000} ; preinsert
  LIN {X 374.916,Y -3131.796,Z -153.095,A 92.55766,B 0.00000,C -180.00000} ; insert
  LIN {X 374.916,Y -3131.796,Z -153.095,A 92.55766,B 0.00000,C -180.00000} ; release
  LIN {X 374.916,Y -3131.796,Z 146.905,A 92.55766,B 0.00000,C -180.00000} ; retreat
  ; Step 1540, bar 2250
  LIN {X -374.916,Y -3131.796,Z 1047.576,A 87.44234,B 0.00000,C 180.00000} ; outside
  LIN {X -374.916,Y -3131.796,Z 96.905,A 87.44234,B 0.00000,C 180.00000} ; preinsert
  LIN {X -374.916,Y -3131.796,Z -153.095,A 87.44234,B 0.00000,C 180.00000} ; insert
  LIN {X -374.916,Y -3131.796,Z -153.095,A 87.44234,B 0.00000,C 180.00000} ; release
  LIN {X -374.916,Y -3131.796,Z 146.905,A 87.44234,B 0.00000,C 180.00000} ; retreat
  ; Step 1541, bar 2256
  LIN {X -1124.916,Y -3131.796,Z 1047.576,A 87.44234,B 0.00000,C 180.00000} ; outside
  LIN {X -1124.916,Y -3131.796,Z 96.905,A 87.44234,B 0.00000,C 180.00000} ; preinsert
  LIN {X -1124.916,Y -3131.796,Z -153.095,A 87.44234,B 0.00000,C 180.00000} ; insert
  LIN {X -1124.916,Y -3131.796,Z -153.095,A 87.44234,B 0.00000,C 180.00000} ; release
  LIN {X -1124.916,Y -3131.796,Z 146.905,A 87.44234,B 0.00000,C 180.00000} ; retreat
  ; Step 1542, bar 2262
  LIN {X -1874.916,Y -3131.796,Z 1047.576,A 87.44234,B 0.00000,C 180.00000} ; outside
  LIN {X -1874.916,Y -3131.796,Z 96.905,A 87.44234,B 0.00000,C 180.00000} ; preinsert
  LIN {X -1874.916,Y -3131.796,Z -153.095,A 87.44234,B 0.00000,C 180.00000} ; insert
  LIN {X -1874.916,Y -3131.796,Z -153.095,A 87.44234,B 0.00000,C 180.00000} ; release
  LIN {X -1874.916,Y -3131.796,Z 146.905,A 87.44234,B 0.00000,C 180.00000} ; retreat
  ; Step 1543, bar 2268
  LIN {X -2624.916,Y -3131.796,Z 1047.576,A 87.44234,B 0.00000,C 180.00000} ; outside
  LIN {X -2624.916,Y -3131.796,Z 96.905,A 87.44234,B 0.00000,C 180.00000} ; preinsert
  LIN {X -2624.916,Y -3131.796,Z -153.095,A 87.44234,B 0.00000,C 180.00000} ; insert
  LIN {X -2624.916,Y -3131.796,Z -153.095,A 87.44234,B 0.00000,C 180.00000} ; release
  LIN {X -2624.916,Y -3131.796,Z 146.905,A 87.44234,B 0.00000,C 180.00000} ; retreat
  ; Step 1544, bar 2274
  LIN {X -3374.916,Y -3131.796,Z 1047.576,A 87.44234,B 0.00000,C 180.00000} ; outside
  LIN {X -3374.916,Y -3131.796,Z 96.905,A 87.44234,B 0.00000,C 180.00000} ; preinsert
  LIN {X -3374.916,Y -3131.796,Z -153.095,A 87.44234,B 0.00000,C 180.00000} ; insert
  LIN {X -3374.916,Y -3131.796,Z -153.095,A 87.44234,B 0.00000,C 180.00000} ; release
  LIN {X -3374.916,Y -3131.796,Z 146.905,A 87.44234,B 0.00000,C 180.00000} ; retreat
  ; Step 1545, bar 2280
  LIN {X -4124.916,Y -3131.796,Z 1047.576,A 87.44234,B 0.00000,C -180.00000} ; outside
  LIN {X -4124.916,Y -3131.796,Z 96.905,A 87.44234,B 0.00000,C -180.00000} ; preinsert
  LIN {X -4124.916,Y -3131.796,Z -153.095,A 87.44234,B 0.00000,C -180.00000} ; insert
  LIN {X -4124.916,Y -3131.796,Z -153.095,A 87.44234,B 0.00000,C -180.00000} ; release
  LIN {X -4124.916,Y -3131.796,Z 146.905,A 87.44234,B 0.00000,C -180.00000} ; retreat
  ; Step 1546, bar 2286
  LIN {X -4874.916,Y -3131.796,Z 1047.576,A 87.44234,B 0.00000,C -180.00000} ; outside
  LIN {X -4874.916,Y -3131.796,Z 96.905,A 87.44234,B 0.00000,C -180.00000} ; preinsert
  LIN {X -4874.916,Y -3131.796,Z -153.095,A 87.44234,B 0.00000,C -180.00000} ; insert
  LIN {X -4874.916,Y -3131.796,Z -153.095,A 87.44234,B 0.00000,C -180.00000} ; release
  LIN {X -4874.916,Y -3131.796,Z 146.905,A 87.44234,B 0.00000,C -180.00000} ; retreat
  ; Step 1547, bar 2292
  LIN {X -5624.916,Y -3131.796,Z 1047.576,A 87.44234,B 0.00000,C -180.00000} ; outside
  LIN {X -5624.916,Y -3131.796,Z 96.905,A 87.44234,B 0.00000,C -180.00000} ; preinsert
  LIN {X -5624.916,Y -3131.796,Z -153.095,A 87.44234,B 0.00000,C -180.00000} ; insert
  LIN {X -5624.916,Y -3131.796,Z -153.095,A 87.44234,B 0.00000,C -180.00000} ; release
  LIN {X -5624.916,Y -3131.796,Z 146.905,A 87.44234,B 0.00000,C -180.00000} ; retreat
  ; Step 1548, bar 2298
  LIN {X -6374.916,Y -3131.796,Z 1047.576,A 87.44234,B 0.00000,C -180.00000} ; outside
  LIN {X -6374.916,Y -3131.796,Z 96.905,A 87.44234,B 0.00000,C -180.00000} ; preinsert
  LIN {X -6374.916,Y -3131.796,Z -153.095,A 87.44234,B 0.00000,C -180.00000} ; insert
  LIN {X -6374.916,Y -3131.796,Z -153.095,A 87.44234,B 0.00000,C -180.00000} ; release
  LIN {X -6374.916,Y -3131.796,Z 146.905,A 87.44234,B 0.00000,C -180.00000} ; retreat
  ; Step 1549, bar 2304
  LIN {X -7124.916,Y -3131.796,Z 1047.576,A 87.44234,B 0.00000,C -180.00000} ; outside
  LIN {X -7124.916,Y -3131.796,Z 96.905,A 87.44234,B 0.00000,C -180.00000} ; preinsert
  LIN {X -7124.916,Y -3131.796,Z -153.095,A 87.44234,B 0.00000,C -180.00000} ; insert
  LIN {X -7124.916,Y -3131.796,Z -153.095,A 87.44234,B 0.00000,C -180.00000} ; release
  LIN {X -7124.916,Y -3131.796,Z 146.905,A 87.44234,B 0.00000,C -180.00000} ; retreat
  ; Step 1550, bar 2310
  LIN {X -7874.916,Y -3131.796,Z 1047.576,A 87.44234,B 0.00000,C -180.00000} ; outside
  LIN {X -7874.916,Y -3131.796,Z 96.905,A 87.44234,B 0.00000,C -180.00000} ; preinsert
  LIN {X -7874.916,Y -3131.796,Z -153.095,A 87.44234,B 0.00000,C -180.00000} ; insert
  LIN {X -7874.916,Y -3131.796,Z -153.095,A 87.44234,B 0.00000,C -180.00000} ; release
  LIN {X -7874.916,Y -3131.796,Z 146.905,A 87.44234,B 0.00000,C -180.00000} ; retreat
  ; Step 1551, bar 2316
  LIN {X -8624.916,Y -3131.796,Z 1047.576,A 87.44234,B 0.00000,C 180.00000} ; outside
  LIN {X -8624.916,Y -3131.796,Z 96.905,A 87.44234,B 0.00000,C 180.00000} ; preinsert
  LIN {X -8624.916,Y -3131.796,Z -153.095,A 87.44234,B 0.00000,C 180.00000} ; insert
  LIN {X -8624.916,Y -3131.796,Z -153.095,A 87.44234,B 0.00000,C 180.00000} ; release
  LIN {X -8624.916,Y -3131.796,Z 146.905,A 87.44234,B 0.00000,C 180.00000} ; retreat
  ; Step 1552, bar 2322
  LIN {X -9374.916,Y -3131.796,Z 1047.576,A 87.44234,B 0.00000,C 180.00000} ; outside
  LIN {X -9374.916,Y -3131.796,Z 96.905,A 87.44234,B 0.00000,C 180.00000} ; preinsert
  LIN {X -9374.916,Y -3131.796,Z -153.095,A 87.44234,B 0.00000,C 180.00000} ; insert
  LIN {X -9374.916,Y -3131.796,Z -153.095,A 87.44234,B 0.00000,C 180.00000} ; release
  LIN {X -9374.916,Y -3131.796,Z 146.905,A 87.44234,B 0.00000,C 180.00000} ; retreat
  ; Step 1553, bar 2328
  LIN {X -10124.916,Y -3131.796,Z 1047.576,A 87.44234,B 0.00000,C 180.00000} ; outside
  LIN {X -10124.916,Y -3131.796,Z 96.905,A 87.44234,B 0.00000,C 180.00000} ; preinsert
  LIN {X -10124.916,Y -3131.796,Z -153.095,A 87.44234,B 0.00000,C 180.00000} ; insert
  LIN {X -10124.916,Y -3131.796,Z -153.095,A 87.44234,B 0.00000,C 180.00000} ; release
  LIN {X -10124.916,Y -3131.796,Z 146.905,A 87.44234,B 0.00000,C 180.00000} ; retreat
  ; Step 1554, bar 2334
  LIN {X -10874.916,Y -3131.796,Z 1047.576,A 87.44234,B 0.00000,C 180.00000} ; outside
  LIN {X -10874.916,Y -3131.796,Z 96.905,A 87.44234,B 0.00000,C 180.00000} ; preinsert
  LIN {X -10874.916,Y -3131.796,Z -153.095,A 87.44234,B 0.00000,C 180.00000} ; insert
  LIN {X -10874.916,Y -3131.796,Z -153.095,A 87.44234,B 0.00000,C 180.00000} ; release
  LIN {X -10874.916,Y -3131.796,Z 146.905,A 87.44234,B 0.00000,C 180.00000} ; retreat
  ; Step 1555, bar 2340
  LIN {X -11624.916,Y -3131.796,Z 1047.576,A 87.44234,B 0.00000,C 180.00000} ; outside
  LIN {X -11624.916,Y -3131.796,Z 96.905,A 87.44234,B 0.00000,C 180.00000} ; preinsert
  LIN {X -11624.916,Y -3131.796,Z -153.095,A 87.44234,B 0.00000,C 180.00000} ; insert
  LIN {X -11624.916,Y -3131.796,Z -153.095,A 87.44234,B 0.00000,C 180.00000} ; release
  LIN {X -11624.916,Y -3131.796,Z 146.905,A 87.44234,B 0.00000,C 180.00000} ; retreat
  ; Step 1556, bar 2346
  LIN {X -12249.916,Y -3131.796,Z 1047.576,A 87.44234,B 0.00000,C 180.00000} ; outside
  LIN {X -12249.916,Y -3131.796,Z 96.905,A 87.44234,B 0.00000,C 180.00000} ; preinsert
  LIN {X -12249.916,Y -3131.796,Z -153.095,A 87.44234,B 0.00000,C 180.00000} ; insert
  LIN {X -12249.916,Y -3131.796,Z -153.095,A 87.44234,B 0.00000,C 180.00000} ; release
  LIN {X -12249.916,Y -3131.796,Z 146.905,A 87.44234,B 0.00000,C 180.00000} ; retreat
  ; Step 1557, bar 2354
  LIN {X -12849.916,Y -3131.796,Z 1047.576,A 87.44234,B 0.00000,C 180.00000} ; outside
  LIN {X -12849.916,Y -3131.796,Z 96.905,A 87.44234,B 0.00000,C 180.00000} ; preinsert
  LIN {X -12849.916,Y -3131.796,Z -153.095,A 87.44234,B 0.00000,C 180.00000} ; insert
  LIN {X -12849.916,Y -3131.796,Z -153.095,A 87.44234,B 0.00000,C 180.00000} ; release
  LIN {X -12849.916,Y -3131.796,Z 146.905,A 87.44234,B 0.00000,C 180.00000} ; retreat
  ; Step 1558, bar 2360
  LIN {X -13449.916,Y -3131.796,Z 1047.576,A 87.44234,B 0.00000,C 180.00000} ; outside
  LIN {X -13449.916,Y -3131.796,Z 96.905,A 87.44234,B 0.00000,C 180.00000} ; preinsert
  LIN {X -13449.916,Y -3131.796,Z -153.095,A 87.44234,B 0.00000,C 180.00000} ; insert
  LIN {X -13449.916,Y -3131.796,Z -153.095,A 87.44234,B 0.00000,C 180.00000} ; release
  LIN {X -13449.916,Y -3131.796,Z 146.905,A 87.44234,B 0.00000,C 180.00000} ; retreat
  ; Step 1559, bar 2366
  LIN {X -14049.916,Y -3131.796,Z 1047.576,A 87.44234,B 0.00000,C 180.00000} ; outside
  LIN {X -14049.916,Y -3131.796,Z 96.905,A 87.44234,B 0.00000,C 180.00000} ; preinsert
  LIN {X -14049.916,Y -3131.796,Z -153.095,A 87.44234,B 0.00000,C 180.00000} ; insert
  LIN {X -14049.916,Y -3131.796,Z -153.095,A 87.44234,B 0.00000,C 180.00000} ; release
  LIN {X -14049.916,Y -3131.796,Z 146.905,A 87.44234,B 0.00000,C 180.00000} ; retreat
  ; Step 1560, bar 2372
  LIN {X -14649.916,Y -3131.796,Z 1047.576,A 87.44234,B 0.00000,C 180.00000} ; outside
  LIN {X -14649.916,Y -3131.796,Z 96.905,A 87.44234,B 0.00000,C 180.00000} ; preinsert
  LIN {X -14649.916,Y -3131.796,Z -153.095,A 87.44234,B 0.00000,C 180.00000} ; insert
  LIN {X -14649.916,Y -3131.796,Z -153.095,A 87.44234,B 0.00000,C 180.00000} ; release
  LIN {X -14649.916,Y -3131.796,Z 146.905,A 87.44234,B 0.00000,C 180.00000} ; retreat
  ; Step 1561, bar 2378
  LIN {X -15249.916,Y -3131.796,Z 1047.576,A 87.44234,B 0.00000,C 180.00000} ; outside
  LIN {X -15249.916,Y -3131.796,Z 96.905,A 87.44234,B 0.00000,C 180.00000} ; preinsert
  LIN {X -15249.916,Y -3131.796,Z -153.095,A 87.44234,B 0.00000,C 180.00000} ; insert
  LIN {X -15249.916,Y -3131.796,Z -153.095,A 87.44234,B 0.00000,C 180.00000} ; release
  LIN {X -15249.916,Y -3131.796,Z 146.905,A 87.44234,B 0.00000,C 180.00000} ; retreat
  ; Step 1562, bar 2384
  LIN {X -15849.916,Y -3131.796,Z 1047.576,A 87.44234,B 0.00000,C 180.00000} ; outside
  LIN {X -15849.916,Y -3131.796,Z 96.905,A 87.44234,B 0.00000,C 180.00000} ; preinsert
  LIN {X -15849.916,Y -3131.796,Z -153.095,A 87.44234,B 0.00000,C 180.00000} ; insert
  LIN {X -15849.916,Y -3131.796,Z -153.095,A 87.44234,B 0.00000,C 180.00000} ; release
  LIN {X -15849.916,Y -3131.796,Z 146.905,A 87.44234,B 0.00000,C 180.00000} ; retreat
  ; Step 1563, bar 2105
  LIN {X -15849.916,Y 3131.796,Z 1047.576,A -87.44234,B 0.00000,C 180.00000} ; outside
  LIN {X -15849.916,Y 3131.796,Z 96.905,A -87.44234,B 0.00000,C 180.00000} ; preinsert
  LIN {X -15849.916,Y 3131.796,Z -153.095,A -87.44234,B 0.00000,C 180.00000} ; insert
  LIN {X -15849.916,Y 3131.796,Z -153.095,A -87.44234,B 0.00000,C 180.00000} ; release
  LIN {X -15849.916,Y 3131.796,Z 146.905,A -87.44234,B 0.00000,C 180.00000} ; retreat
  ; Step 1564, bar 2099
  LIN {X -15249.916,Y 3131.796,Z 1047.576,A -87.44234,B 0.00000,C 180.00000} ; outside
  LIN {X -15249.916,Y 3131.796,Z 96.905,A -87.44234,B 0.00000,C 180.00000} ; preinsert
  LIN {X -15249.916,Y 3131.796,Z -153.095,A -87.44234,B 0.00000,C 180.00000} ; insert
  LIN {X -15249.916,Y 3131.796,Z -153.095,A -87.44234,B 0.00000,C 180.00000} ; release
  LIN {X -15249.916,Y 3131.796,Z 146.905,A -87.44234,B 0.00000,C 180.00000} ; retreat
  ; Step 1565, bar 2093
  LIN {X -14649.916,Y 3131.796,Z 1047.576,A -87.44234,B 0.00000,C 180.00000} ; outside
  LIN {X -14649.916,Y 3131.796,Z 96.905,A -87.44234,B 0.00000,C 180.00000} ; preinsert
  LIN {X -14649.916,Y 3131.796,Z -153.095,A -87.44234,B 0.00000,C 180.00000} ; insert
  LIN {X -14649.916,Y 3131.796,Z -153.095,A -87.44234,B 0.00000,C 180.00000} ; release
  LIN {X -14649.916,Y 3131.796,Z 146.905,A -87.44234,B 0.00000,C 180.00000} ; retreat
  ; Step 1566, bar 2087
  LIN {X -14049.916,Y 3131.796,Z 1047.576,A -87.44234,B 0.00000,C 180.00000} ; outside
  LIN {X -14049.916,Y 3131.796,Z 96.905,A -87.44234,B 0.00000,C 180.00000} ; preinsert
  LIN {X -14049.916,Y 3131.796,Z -153.095,A -87.44234,B 0.00000,C 180.00000} ; insert
  LIN {X -14049.916,Y 3131.796,Z -153.095,A -87.44234,B 0.00000,C 180.00000} ; release
  LIN {X -14049.916,Y 3131.796,Z 146.905,A -87.44234,B 0.00000,C 180.00000} ; retreat
  ; Step 1567, bar 2081
  LIN {X -13449.916,Y 3131.796,Z 1047.576,A -87.44234,B 0.00000,C 180.00000} ; outside
  LIN {X -13449.916,Y 3131.796,Z 96.905,A -87.44234,B 0.00000,C 180.00000} ; preinsert
  LIN {X -13449.916,Y 3131.796,Z -153.095,A -87.44234,B 0.00000,C 180.00000} ; insert
  LIN {X -13449.916,Y 3131.796,Z -153.095,A -87.44234,B 0.00000,C 180.00000} ; release
  LIN {X -13449.916,Y 3131.796,Z 146.905,A -87.44234,B 0.00000,C 180.00000} ; retreat
  ; Step 1568, bar 2075
  LIN {X -12849.916,Y 3131.796,Z 1047.576,A -87.44234,B 0.00000,C 180.00000} ; outside
  LIN {X -12849.916,Y 3131.796,Z 96.905,A -87.44234,B 0.00000,C 180.00000} ; preinsert
  LIN {X -12849.916,Y 3131.796,Z -153.095,A -87.44234,B 0.00000,C 180.00000} ; insert
  LIN {X -12849.916,Y 3131.796,Z -153.095,A -87.44234,B 0.00000,C 180.00000} ; release
  LIN {X -12849.916,Y 3131.796,Z 146.905,A -87.44234,B 0.00000,C 180.00000} ; retreat
  ; Step 1569, bar 2067
  LIN {X -12249.916,Y 3131.796,Z 1047.576,A -87.44234,B 0.00000,C 180.00000} ; outside
  LIN {X -12249.916,Y 3131.796,Z 96.905,A -87.44234,B 0.00000,C 180.00000} ; preinsert
  LIN {X -12249.916,Y 3131.796,Z -153.095,A -87.44234,B 0.00000,C 180.00000} ; insert
  LIN {X -12249.916,Y 3131.796,Z -153.095,A -87.44234,B 0.00000,C 180.00000} ; release
  LIN {X -12249.916,Y 3131.796,Z 146.905,A -87.44234,B 0.00000,C 180.00000} ; retreat
  ; Step 1570, bar 2061
  LIN {X -11624.916,Y 3131.796,Z 1047.576,A -87.44234,B 0.00000,C 180.00000} ; outside
  LIN {X -11624.916,Y 3131.796,Z 96.905,A -87.44234,B 0.00000,C 180.00000} ; preinsert
  LIN {X -11624.916,Y 3131.796,Z -153.095,A -87.44234,B 0.00000,C 180.00000} ; insert
  LIN {X -11624.916,Y 3131.796,Z -153.095,A -87.44234,B 0.00000,C 180.00000} ; release
  LIN {X -11624.916,Y 3131.796,Z 146.905,A -87.44234,B 0.00000,C 180.00000} ; retreat
  ; Step 1571, bar 2055
  LIN {X -10874.916,Y 3131.796,Z 1047.576,A -87.44234,B 0.00000,C 180.00000} ; outside
  LIN {X -10874.916,Y 3131.796,Z 96.905,A -87.44234,B 0.00000,C 180.00000} ; preinsert
